// TIA Portal V20 export
// export: Created 2025-12-01T14:56:30.7058292Z, ExportSetting None, DisplayName Totally Integrated Automation Portal, DisplayVersion V20 Update 3, DisplayName TIA Portal Openness, DisplayVersion V20 Update 3, DisplayName TIA Portal Version Control Interface, DisplayVersion V20 Update 3, DisplayName STEP 7 Professional, DisplayVersion V20 Update 3, DisplayName STEP 7 Safety, DisplayVersion V20 Update 2, DisplayName WinCC Basic/Comfort/Advanced, DisplayVersion V20 Update 3, DisplayName WinCC Professional, DisplayVersion V20 Update 3, DisplayName WinCC Unified, DisplayVersion V20 Update 3
FUNCTION_BLOCK "FB435_CRTL_V_E1_S23_BLOQ_OrdJDT"   // FB435, LAD
TITLE = Control del Ramal de Salidas
{ S7_Optimized_Access := 'FALSE' }
AUTHOR : TLigero
NAME : 20190213
VERSION : 3.3
// stored: AutoNumber false, SetENOAutomatically false
   VAR_INPUT
      Mesa : UInt;   // Número de mesa
      En_Tension : Bool;
      pHsMx_E1 : Bool;   // pHs DE PRESENCIA de la Mesa en E1
      pHsMx_S3 : Bool;   // pHs DE AUSENCIA de la Mesa en S3
      pHsMx_S2 : Bool;   // pHs DE AUSENCIA de la Mesa en S2
      En_Pos_WS_0 : Bool;   // Desviador en posicion 0 grados
      En_Pos_WS_45 : Bool;   // Desviador en posicion de desvio
      Termico_E1S3 : Bool;   // Proteccion del Tx en E1E3
      Avance_Tx_Ent : Bool;   // Avance del Tx de entrada. Primer tramo
      Avance_Tx_Sal : Bool;   // Avance del Tx de Salida por S3 o S2
      PTF_Sal_M3 : Bool;   // S3 >> Mesa Siguiente PTF
      NXT_Avance_S3 : Bool;   // S3 >> Mesa Siguiente avanzando
      PTF_Sal_M2 : Bool;   // S2 >> Mesa Siguiente PTF
      NXT_Avance_S2 : Bool;   // S2 >> Mesa Siguiente avanzando
      F_EnvMens_Mx : Bool;   // Fin de Envio de Mensaje
      Mx_Bloq_Activo : Bool;   // Bloqueo Activo de la Mesa
      MX_FlujoPrin_S2 : Bool;   // El flujo principal es Saliendo por S2
      AVTF_MAnt_Mx : Bool;   // E1 >> Mesa Anterior AVTF
      Habilitar_orden_JDT : Bool := false;   // El JDT tendrá el control del cruce con orden
      Num_Cruce : UInt;   // Número de cruce.
      DB_FIFO_Cruce : UInt := 213;   // DB de la FIFO de ordenes del cruce
      Lng_FIFO_Cruce : UInt := 1;   // Longitut de la FIFO de ordenes del cruce
      Valor_Orden_S2 : Word := 16#81;   // Con que orden entra por S2
      MesaS2 : UInt;   // Número de mesa por S2
      MesaS3 : UInt;   // Número de mesa por S3
      V_CNT_pHsMx : UDInt := 500;   // Valor de Presencia en ms
      V_CNT_ApHsMx : UDInt := 500;   // Valor de Ausencia en ms
      V_Vaciado : UDInt := 5000;   // Valor de vaciado en ms
      V_TOut_Desviador : UDInt := 2000;   // TimeOut de los cilindros del desviador en ms
      V_TOut_Tx_Mx : UDInt := 3000;   // TimeOut de Atasco en ms
      V_CNT_ApHsMx_S3 : UDInt := 500;   // Valor de Ausencia por S3 en ms
      V_CNT_ApHsMx_S2 : UDInt := 500;   // Valor de Ausencia por S2 en ms
      V_Orden_Bloqueo : UDInt := 3000;   // en ms
   END_VAR
   VAR_OUTPUT
      P_EnvMens_PMx : Bool;   // Permiso de Enviar Mensaje de Presencia
      Etiqueta_Jdt : UDInt;   // Etiqueta que ha sido leida
      Orden_Ejecutada_Jdt : UInt;   // Orden que se ha ejecutado
      PTF_MAnt_Mx : Bool;   // E1 >> Mesa Anterior PTF
      AVTF_Sal_M2 : Bool;   // S3 >> Mesa Siguiente AVTF
      NXT_Descarga_Act_S2 : Bool;   // S3 >> Mesa Siguiente descarga activa
      AVTF_Sal_M3 : Bool;   // S3 >> Mesa Siguiente AVTF
      NXT_Descarga_Act_S3 : Bool;   // S3 >> Mesa Siguiente descarga activa
   END_VAR
   VAR
      T1_ET00 : Bool;   // Reset
      T1_ET08 : Bool;
      T1_ET01 : Bool;   // Entrada Vacia
      T1_ET10 : Bool;   // Carga Entrada
      T1_ET02 : Bool;   // Entrada Cargada
      T1_ET03 : Bool;   // Vaciando Entrada
      T1_ET20 : Bool;   // Carga Salida
      T1_ET21 : Bool;   // Salida Vacia
      T1_ET50 : Bool;   // Continuar
      T1_ET60 : Bool;   // Entrar
      T1_ET110 : Bool;   // Extraer orden
      T1_ET111 : Bool;
      T1_ET112 : Bool;
      T1_ET02_JDT : Bool;
      FP_ET2_JDT : Bool;
      FIFO_OK : Bool;
      TRANS_OK : Bool;
      O_Bloqueo : Bool;
      Vaciado_1 : Bool;
      Vaciado_2 : Bool;
      FN_ET20 : Bool;
      MemoPresenciaJdt : Bool;
      Maux_FN_Phs_S2 : Bool;
      mem_fn_phs_s2 : Bool;
      Maux_FN_Phs_S3 : Bool;
      mem_fn_phs_s3 : Bool;
      maux_fp_disparo : Bool;
      maux_fn_phs_e1 : Bool;
      ok_vaciado : Bool;
      CNT_ERR_PHS : Int;
      CNT_pHs_WS : UDInt;
      CNT_Aus_WS : UDInt;
      CNT_aus_ent : UDInt;
      CNT_aus_cont : UDInt;
      CNT_bloqueo : UDInt;
      TIMV_WS : UDInt;
      TMP_Err_Pist_pos_0 : UDInt;
      TMP_Paro : UDInt;
      TMP_Err_Pist_pos_45 : UDInt;
      TMP_Err_Tout_avance_E : UDInt;
      TMP_Err_Tout_avance_S : UDInt;
      TMP_En_Tension : UDInt;
      Datos_Scanner { S7_SetPoint := 'True'} : "ROUT_Orden_Fifo_Scanner";
   END_VAR
   VAR_TEMP
      EstadoZona : "EstadoZona";   // Estado de Zona de la Mesa
      EstadoVI : "EstadosMesa";   // Estado del Vehiculo Inteliguente de la Mesa
      ConfigFB : "UDT_ConfigFB";   // Configuracion de la FB de la Mesa
      TEMP_ET00 : Bool;
      O_Continuar : Bool;
      O_Entrar : Bool;
      O_Vaciar : Bool;
      cnt_phs_ok : Bool;
      cnt_aus_ok : Bool;
      OK_Aus_Entrar : Bool;
      OK_Aus_Cont : Bool;
      timeout_piston : Bool;
      ok_tension : Bool;
      Aux_W_Moti : Word;
      Moti_INIC : Bool;
      Moti_ERRO : Bool;
      Moti_NENC : Bool;
      Moti_NORM : Bool;
      ok_bloqueo : Bool;
      O_Continuar_JDT : Bool;
      O_Entrar_JDT : Bool;
      atasco : Bool;
      t_paro : Bool;
      I_V_Ord_Entrar : UInt;
      I_Ord_Filtrada : UInt;
      INT_ORDEN : UInt;
      Aux_W_Orden : Word;
   END_VAR
   VAR_TEMP   // added for the SCL form of the ladder/FBD networks
      _w1 : Bool;
      _w2 : Bool;
      _w3 : Bool;
      _w4 : Bool;
      _w5 : Bool;
      _w6 : Bool;
      _w7 : Bool;
   END_VAR
BEGIN

REGION Network 1: INICIALIZAR - Recoger las Variables de Estado de la Mesa
   // Se recoge - Estado_CBx
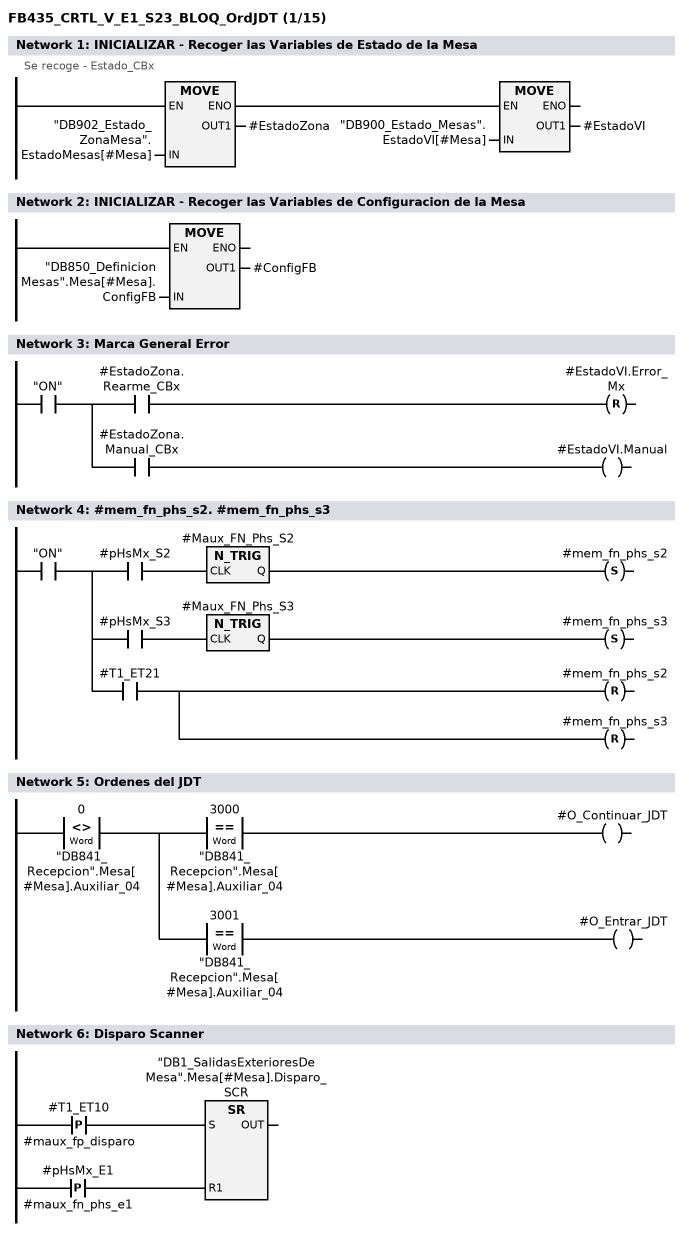
   RUNG wire#powerrail
      Move(in := "DB902_Estado_ZonaMesa".EstadoMesas[#Mesa], out1 => #EstadoZona)
      Move(in := "DB900_Estado_Mesas".EstadoVI[#Mesa], out1 => #EstadoVI)
   END_RUNG
   // the same network as SCL:
   #EstadoZona := "DB902_Estado_ZonaMesa".EstadoMesas[#Mesa];
   #EstadoVI := "DB900_Estado_Mesas".EstadoVI[#Mesa];
END_REGION

REGION Network 2: INICIALIZAR - Recoger las Variables de Configuracion de la Mesa
   RUNG wire#powerrail
      Move(in := "DB850_DefinicionMesas".Mesa[#Mesa].ConfigFB, out1 => #ConfigFB)
   END_RUNG
   // the same network as SCL:
   #ConfigFB := "DB850_DefinicionMesas".Mesa[#Mesa].ConfigFB;
END_REGION

REGION Network 3: Marca General Error
   RUNG wire#powerrail
      Contact( "ON" )
      wire#w1
      Contact( #EstadoZona.Rearme_CBx )
      R_Coil( #EstadoVI.Error_Mx )
   END_RUNG
   RUNG wire#w1
      Contact( #EstadoZona.Manual_CBx )
      Coil( #EstadoVI.Manual )
   END_RUNG
   // the same network as SCL:
   IF "ON" AND #EstadoZona.Rearme_CBx THEN #EstadoVI.Error_Mx := FALSE; END_IF;
   #EstadoVI.Manual := "ON" AND #EstadoZona.Manual_CBx;
END_REGION

REGION Network 4: #mem_fn_phs_s2. #mem_fn_phs_s3
   RUNG wire#powerrail
      Contact( "ON" )
      wire#w1
      Contact( #pHsMx_S2 )
      N_Trig( #Maux_FN_Phs_S2 )
      S_Coil( #mem_fn_phs_s2 )
   END_RUNG
   RUNG wire#w1
      Contact( #pHsMx_S3 )
      N_Trig( #Maux_FN_Phs_S3 )
      S_Coil( #mem_fn_phs_s3 )
   END_RUNG
   RUNG wire#w1
      Contact( #T1_ET21 )
      wire#w2
      R_Coil( #mem_fn_phs_s2 )
   END_RUNG
   RUNG wire#w2
      R_Coil( #mem_fn_phs_s3 )
   END_RUNG
   // the same network as SCL:
   #_w1 := "ON" AND #pHsMx_S2;
   #_w2 := NOT #_w1 AND #Maux_FN_Phs_S2;   // falling edge
   #Maux_FN_Phs_S2 := #_w1;
   IF #_w2 THEN #mem_fn_phs_s2 := TRUE; END_IF;
   #_w3 := "ON" AND #pHsMx_S3;
   #_w4 := NOT #_w3 AND #Maux_FN_Phs_S3;   // falling edge
   #Maux_FN_Phs_S3 := #_w3;
   IF #_w4 THEN #mem_fn_phs_s3 := TRUE; END_IF;
   IF "ON" AND #T1_ET21 THEN
       #mem_fn_phs_s2 := FALSE;
       #mem_fn_phs_s3 := FALSE;
   END_IF;
END_REGION

REGION Network 5: Ordenes del JDT
   RUNG wire#powerrail
      { S7_Templates := "SrcType := Word" } NE_Contact(in1 := 0, in2 := "DB841_Recepcion".Mesa[#Mesa].Auxiliar_04)
      wire#w1
      { S7_Templates := "SrcType := Word" } EQ_Contact(in1 := 3000, in2 := "DB841_Recepcion".Mesa[#Mesa].Auxiliar_04)
      Coil( #O_Continuar_JDT )
   END_RUNG
   RUNG wire#w1
      { S7_Templates := "SrcType := Word" } EQ_Contact(in1 := 3001, in2 := "DB841_Recepcion".Mesa[#Mesa].Auxiliar_04)
      Coil( #O_Entrar_JDT )
   END_RUNG
   // the same network as SCL:
   #_w1 := 0 <> "DB841_Recepcion".Mesa[#Mesa].Auxiliar_04;
   #O_Continuar_JDT := #_w1 AND (3000 = "DB841_Recepcion".Mesa[#Mesa].Auxiliar_04);
   #O_Entrar_JDT := #_w1 AND (3001 = "DB841_Recepcion".Mesa[#Mesa].Auxiliar_04);
END_REGION

REGION Network 6: Disparo Scanner
   RUNG wire#powerrail
      P_Contact(operand := #T1_ET10, bit := #maux_fp_disparo)
      S_SR(operand := "DB1_SalidasExterioresDeMesa".Mesa[#Mesa].Disparo_SCR, r1 := wire#w1)
   END_RUNG
   RUNG wire#powerrail
      P_Contact(operand := #pHsMx_E1, bit := #maux_fn_phs_e1)
   END_RUNG wire#w1
   // the same network as SCL:
   #_w1 := #T1_ET10 AND NOT #maux_fp_disparo;   // rising edge of #T1_ET10
   #maux_fp_disparo := #T1_ET10;
   #_w2 := #pHsMx_E1 AND NOT #maux_fn_phs_e1;   // rising edge of #pHsMx_E1
   #maux_fn_phs_e1 := #pHsMx_E1;
   IF #_w1 THEN
       "DB1_SalidasExterioresDeMesa".Mesa[#Mesa].Disparo_SCR := TRUE;   // SR flip-flop
   END_IF;
   IF #_w2 THEN "DB1_SalidasExterioresDeMesa".Mesa[#Mesa].Disparo_SCR := FALSE; END_IF;
END_REGION

REGION Network 7: GESTION FORZAR ORDENES VACIADO ZONA
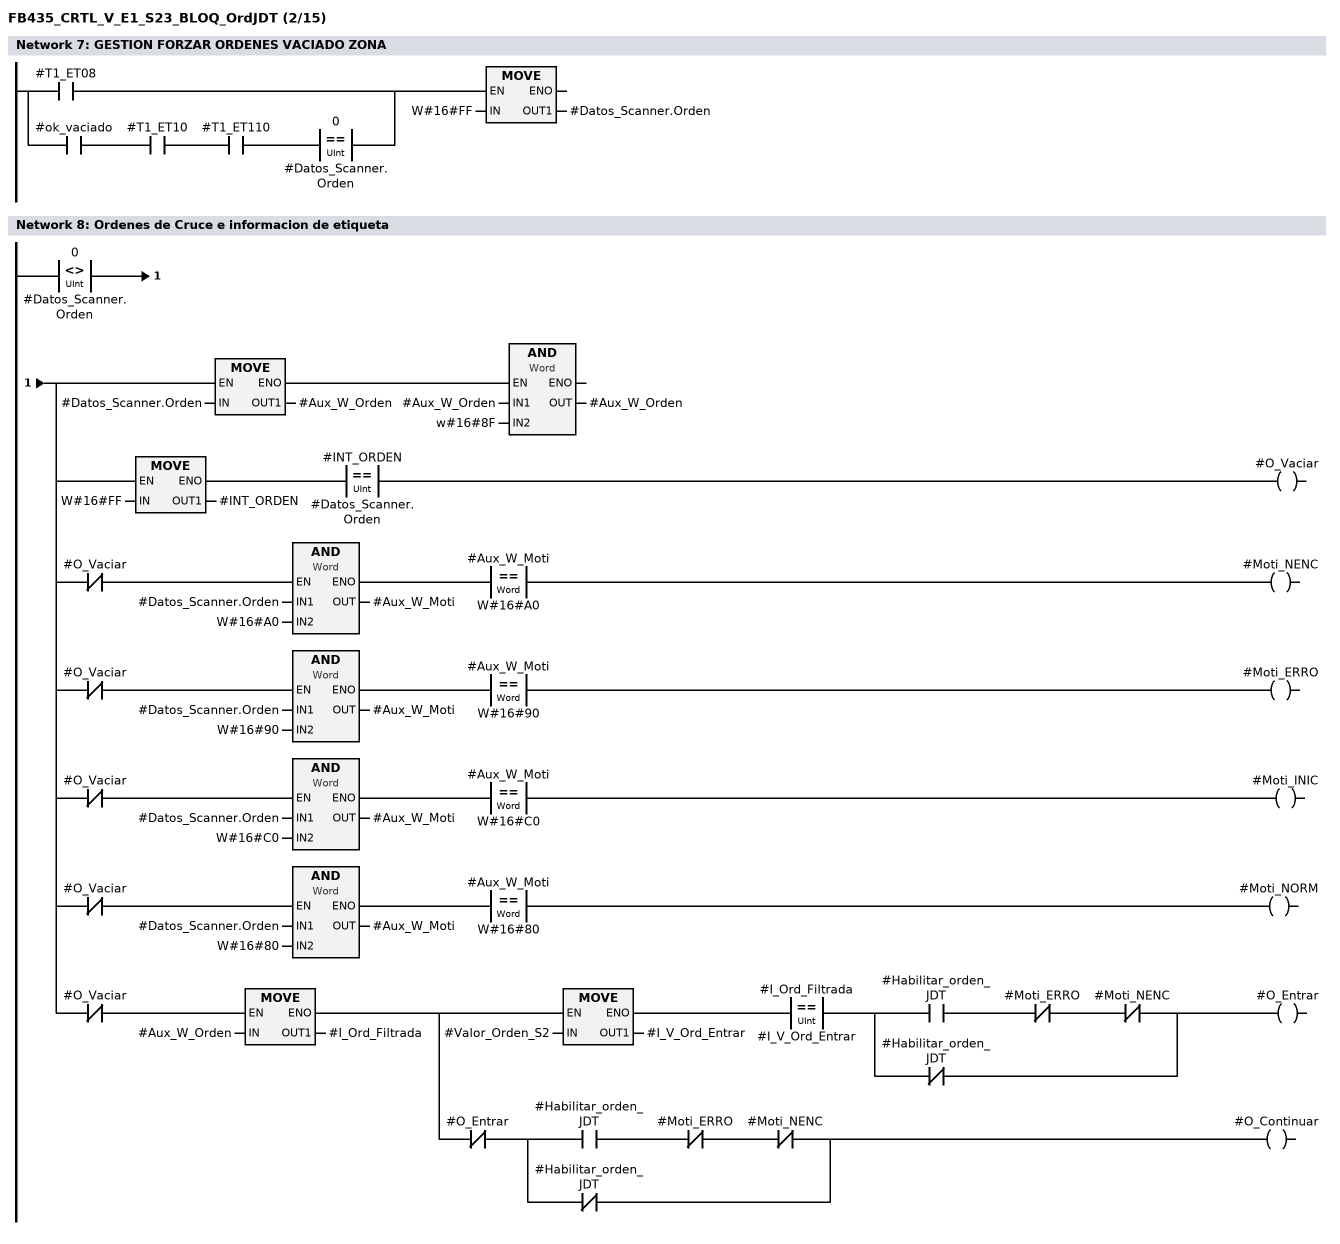
   RUNG wire#powerrail
      Contact( #T1_ET08 )
      wire#w1
      { S7_GenerateENO := "TRUE" } Move(in := W#16#FF, out1 => #Datos_Scanner.Orden)
   END_RUNG
   RUNG wire#powerrail
      Contact( #ok_vaciado )
      Contact( #T1_ET10 )
      Contact( #T1_ET110 )
      { S7_Templates := "SrcType := UInt" } EQ_Contact(in1 := 0, in2 := #Datos_Scanner.Orden)
   END_RUNG wire#w1
   // the same network as SCL:
   IF #T1_ET08 OR (#ok_vaciado AND #T1_ET10 AND #T1_ET110 AND (0 = #Datos_Scanner.Orden)) THEN
       #Datos_Scanner.Orden := W#16#FF;
   END_IF;
END_REGION

REGION Network 8: Ordenes de Cruce e informacion de etiqueta
   RUNG wire#powerrail
      { S7_Templates := "SrcType := UInt" } NE_Contact(in1 := 0, in2 := #Datos_Scanner.Orden)
      wire#w1
      { S7_GenerateENO := "TRUE" } Move(in := #Datos_Scanner.Orden, out1 => #Aux_W_Orden)
      { S7_Templates := "SrcType := Word"; S7_GenerateENO := "TRUE" } And(in1 := #Aux_W_Orden, in2 := w#16#8F, out => #Aux_W_Orden)
   END_RUNG
   RUNG wire#w1
      { S7_GenerateENO := "TRUE" } Move(in := W#16#FF, out1 => #INT_ORDEN)
      { S7_Templates := "SrcType := UInt" } EQ_Contact(in1 := #INT_ORDEN, in2 := #Datos_Scanner.Orden)
      Coil( #O_Vaciar )
   END_RUNG
   RUNG wire#w1
      I_Contact( #O_Vaciar )
      { S7_Templates := "SrcType := Word"; S7_GenerateENO := "TRUE" } And(in1 := #Datos_Scanner.Orden, in2 := W#16#A0, out => #Aux_W_Moti)
      { S7_Templates := "SrcType := Word" } EQ_Contact(in1 := #Aux_W_Moti, in2 := W#16#A0)
      Coil( #Moti_NENC )
   END_RUNG
   RUNG wire#w1
      I_Contact( #O_Vaciar )
      { S7_Templates := "SrcType := Word"; S7_GenerateENO := "TRUE" } And(in1 := #Datos_Scanner.Orden, in2 := W#16#90, out => #Aux_W_Moti)
      { S7_Templates := "SrcType := Word" } EQ_Contact(in1 := #Aux_W_Moti, in2 := W#16#90)
      Coil( #Moti_ERRO )
   END_RUNG
   RUNG wire#w1
      I_Contact( #O_Vaciar )
      { S7_Templates := "SrcType := Word"; S7_GenerateENO := "TRUE" } And(in1 := #Datos_Scanner.Orden, in2 := W#16#C0, out => #Aux_W_Moti)
      { S7_Templates := "SrcType := Word" } EQ_Contact(in1 := #Aux_W_Moti, in2 := W#16#C0)
      Coil( #Moti_INIC )
   END_RUNG
   RUNG wire#w1
      I_Contact( #O_Vaciar )
      { S7_Templates := "SrcType := Word"; S7_GenerateENO := "TRUE" } And(in1 := #Datos_Scanner.Orden, in2 := W#16#80, out => #Aux_W_Moti)
      { S7_Templates := "SrcType := Word" } EQ_Contact(in1 := #Aux_W_Moti, in2 := W#16#80)
      Coil( #Moti_NORM )
   END_RUNG
   RUNG wire#w1
      I_Contact( #O_Vaciar )
      { S7_GenerateENO := "TRUE" } Move(in := #Aux_W_Orden, out1 => #I_Ord_Filtrada)
      wire#w2
      { S7_GenerateENO := "TRUE" } Move(in := #Valor_Orden_S2, out1 => #I_V_Ord_Entrar)
      { S7_Templates := "SrcType := UInt" } EQ_Contact(in1 := #I_Ord_Filtrada, in2 := #I_V_Ord_Entrar)
      wire#w3
      Contact( #Habilitar_orden_JDT )
      I_Contact( #Moti_ERRO )
      I_Contact( #Moti_NENC )
      wire#w4
      Coil( #O_Entrar )
   END_RUNG
   RUNG wire#w3
      I_Contact( #Habilitar_orden_JDT )
   END_RUNG wire#w4
   RUNG wire#w2
      I_Contact( #O_Entrar )
      wire#w5
      Contact( #Habilitar_orden_JDT )
      I_Contact( #Moti_ERRO )
      I_Contact( #Moti_NENC )
      wire#w6
      Coil( #O_Continuar )
   END_RUNG
   RUNG wire#w5
      I_Contact( #Habilitar_orden_JDT )
   END_RUNG wire#w6
   // the same network as SCL:
   // ENO of a box is taken as its EN; it also drops when the box reports an error
   #_w1 := 0 <> #Datos_Scanner.Orden;
   IF #_w1 THEN
       #Aux_W_Orden := #Datos_Scanner.Orden;
       #Aux_W_Orden := #Aux_W_Orden AND w#16#8F;
       #INT_ORDEN := W#16#FF;
   END_IF;
   #O_Vaciar := #_w1 AND (#INT_ORDEN = #Datos_Scanner.Orden);
   #_w2 := #_w1 AND NOT #O_Vaciar;
   IF #_w2 THEN #Aux_W_Moti := #Datos_Scanner.Orden AND W#16#A0; END_IF;
   #Moti_NENC := #_w2 AND (#Aux_W_Moti = W#16#A0);
   #_w3 := #_w1 AND NOT #O_Vaciar;
   IF #_w3 THEN #Aux_W_Moti := #Datos_Scanner.Orden AND W#16#90; END_IF;
   #Moti_ERRO := #_w3 AND (#Aux_W_Moti = W#16#90);
   #_w4 := #_w1 AND NOT #O_Vaciar;
   IF #_w4 THEN #Aux_W_Moti := #Datos_Scanner.Orden AND W#16#C0; END_IF;
   #Moti_INIC := #_w4 AND (#Aux_W_Moti = W#16#C0);
   #_w5 := #_w1 AND NOT #O_Vaciar;
   IF #_w5 THEN #Aux_W_Moti := #Datos_Scanner.Orden AND W#16#80; END_IF;
   #Moti_NORM := #_w5 AND (#Aux_W_Moti = W#16#80);
   #_w6 := #_w1 AND NOT #O_Vaciar;
   IF #_w6 THEN
       #I_Ord_Filtrada := #Aux_W_Orden;
       #I_V_Ord_Entrar := #Valor_Orden_S2;
   END_IF;
   #O_Entrar := #_w6 AND (#I_Ord_Filtrada = #I_V_Ord_Entrar) AND ((#Habilitar_orden_JDT AND NOT #Moti_ERRO AND NOT #Moti_NENC) OR NOT #Habilitar_orden_JDT);
   #O_Continuar := #_w6 AND NOT #O_Entrar AND ((#Habilitar_orden_JDT AND NOT #Moti_ERRO AND NOT #Moti_NENC) OR NOT #Habilitar_orden_JDT);
END_REGION

REGION Network 9: FC912. #V_CNTpHsWS
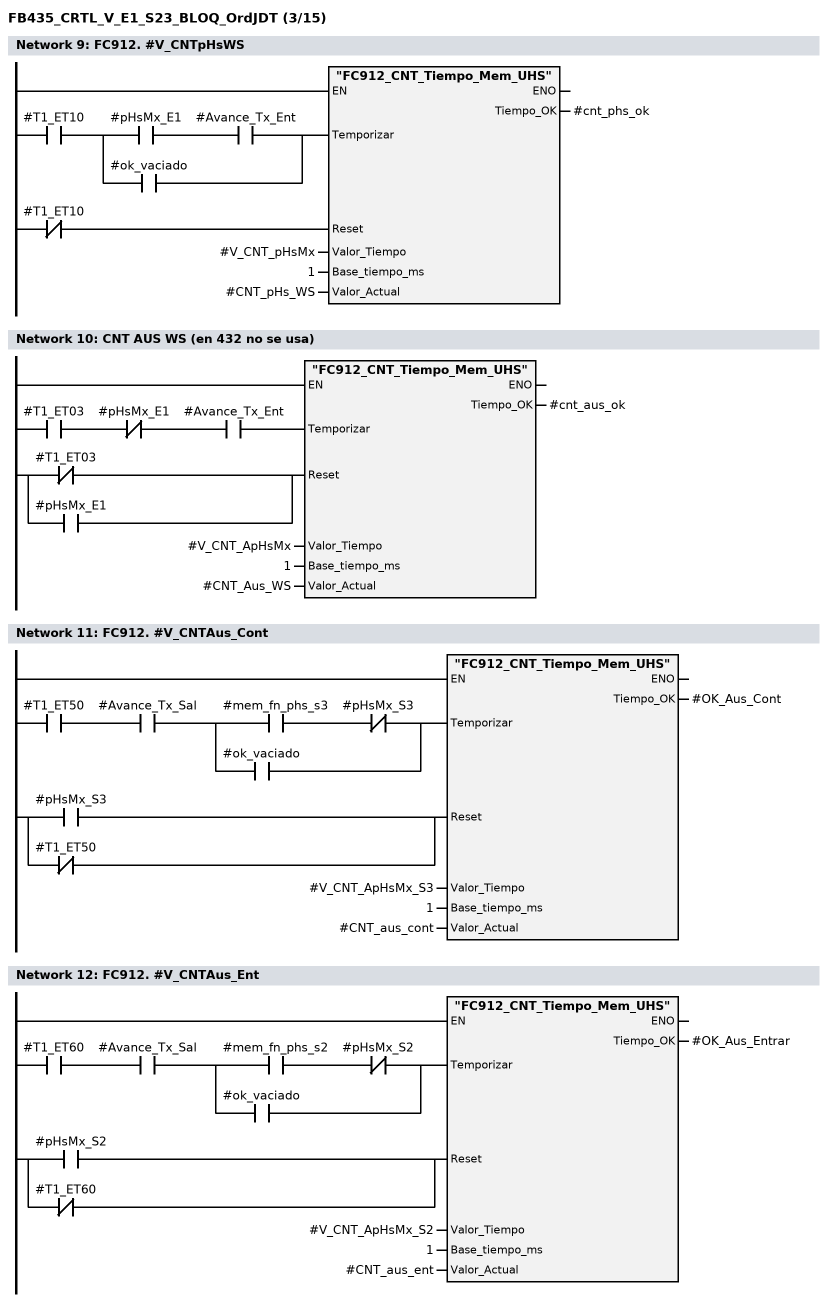
   RUNG wire#powerrail
      "FC912_CNT_Tiempo_Mem_UHS"(Temporizar := wire#w2, Reset := wire#w3, Valor_Tiempo := #V_CNT_pHsMx, Base_tiempo_ms := 1, Valor_Actual := #CNT_pHs_WS, Tiempo_OK => #cnt_phs_ok)
   END_RUNG
   RUNG wire#powerrail
      Contact( #T1_ET10 )
      wire#w1
      Contact( #pHsMx_E1 )
      Contact( #Avance_Tx_Ent )
   END_RUNG wire#w2
   RUNG wire#w1
      Contact( #ok_vaciado )
   END_RUNG wire#w2
   RUNG wire#powerrail
      I_Contact( #T1_ET10 )
   END_RUNG wire#w3
   // the same network as SCL:
   "FC912_CNT_Tiempo_Mem_UHS"(Temporizar := #T1_ET10 AND ((#pHsMx_E1 AND #Avance_Tx_Ent) OR #ok_vaciado),
                           Reset := NOT #T1_ET10,
                           Valor_Tiempo := #V_CNT_pHsMx,
                           Base_tiempo_ms := 1,
                           Valor_Actual := #CNT_pHs_WS,
                           Tiempo_OK => #cnt_phs_ok);
END_REGION

REGION Network 10: CNT AUS WS (en 432 no se usa)
   RUNG wire#powerrail
      "FC912_CNT_Tiempo_Mem_UHS"(Temporizar := wire#w1, Reset := wire#w2, Valor_Tiempo := #V_CNT_ApHsMx, Base_tiempo_ms := 1, Valor_Actual := #CNT_Aus_WS, Tiempo_OK => #cnt_aus_ok)
   END_RUNG
   RUNG wire#powerrail
      Contact( #T1_ET03 )
      I_Contact( #pHsMx_E1 )
      Contact( #Avance_Tx_Ent )
   END_RUNG wire#w1
   RUNG wire#powerrail
      I_Contact( #T1_ET03 )
   END_RUNG wire#w2
   RUNG wire#powerrail
      Contact( #pHsMx_E1 )
   END_RUNG wire#w2
   // the same network as SCL:
   "FC912_CNT_Tiempo_Mem_UHS"(Temporizar := #T1_ET03 AND NOT #pHsMx_E1 AND #Avance_Tx_Ent,
                           Reset := NOT #T1_ET03 OR #pHsMx_E1,
                           Valor_Tiempo := #V_CNT_ApHsMx,
                           Base_tiempo_ms := 1,
                           Valor_Actual := #CNT_Aus_WS,
                           Tiempo_OK => #cnt_aus_ok);
END_REGION

REGION Network 11: FC912. #V_CNTAus_Cont
   RUNG wire#powerrail
      "FC912_CNT_Tiempo_Mem_UHS"(Temporizar := wire#w2, Reset := wire#w3, Valor_Tiempo := #V_CNT_ApHsMx_S3, Base_tiempo_ms := 1, Valor_Actual := #CNT_aus_cont, Tiempo_OK => #OK_Aus_Cont)
   END_RUNG
   RUNG wire#powerrail
      Contact( #T1_ET50 )
      Contact( #Avance_Tx_Sal )
      wire#w1
      Contact( #mem_fn_phs_s3 )
      I_Contact( #pHsMx_S3 )
   END_RUNG wire#w2
   RUNG wire#w1
      Contact( #ok_vaciado )
   END_RUNG wire#w2
   RUNG wire#powerrail
      Contact( #pHsMx_S3 )
   END_RUNG wire#w3
   RUNG wire#powerrail
      I_Contact( #T1_ET50 )
   END_RUNG wire#w3
   // the same network as SCL:
   "FC912_CNT_Tiempo_Mem_UHS"(Temporizar := #T1_ET50 AND #Avance_Tx_Sal AND ((#mem_fn_phs_s3 AND NOT #pHsMx_S3) OR #ok_vaciado),
                           Reset := #pHsMx_S3 OR NOT #T1_ET50,
                           Valor_Tiempo := #V_CNT_ApHsMx_S3,
                           Base_tiempo_ms := 1,
                           Valor_Actual := #CNT_aus_cont,
                           Tiempo_OK => #OK_Aus_Cont);
END_REGION

REGION Network 12: FC912. #V_CNTAus_Ent
   RUNG wire#powerrail
      "FC912_CNT_Tiempo_Mem_UHS"(Temporizar := wire#w2, Reset := wire#w3, Valor_Tiempo := #V_CNT_ApHsMx_S2, Base_tiempo_ms := 1, Valor_Actual := #CNT_aus_ent, Tiempo_OK => #OK_Aus_Entrar)
   END_RUNG
   RUNG wire#powerrail
      Contact( #T1_ET60 )
      Contact( #Avance_Tx_Sal )
      wire#w1
      Contact( #mem_fn_phs_s2 )
      I_Contact( #pHsMx_S2 )
   END_RUNG wire#w2
   RUNG wire#w1
      Contact( #ok_vaciado )
   END_RUNG wire#w2
   RUNG wire#powerrail
      Contact( #pHsMx_S2 )
   END_RUNG wire#w3
   RUNG wire#powerrail
      I_Contact( #T1_ET60 )
   END_RUNG wire#w3
   // the same network as SCL:
   "FC912_CNT_Tiempo_Mem_UHS"(Temporizar := #T1_ET60 AND #Avance_Tx_Sal AND ((#mem_fn_phs_s2 AND NOT #pHsMx_S2) OR #ok_vaciado),
                           Reset := #pHsMx_S2 OR NOT #T1_ET60,
                           Valor_Tiempo := #V_CNT_ApHsMx_S2,
                           Base_tiempo_ms := 1,
                           Valor_Actual := #CNT_aus_ent,
                           Tiempo_OK => #OK_Aus_Entrar);
END_REGION

REGION Network 13: FC912. #V_TmpBloqueo
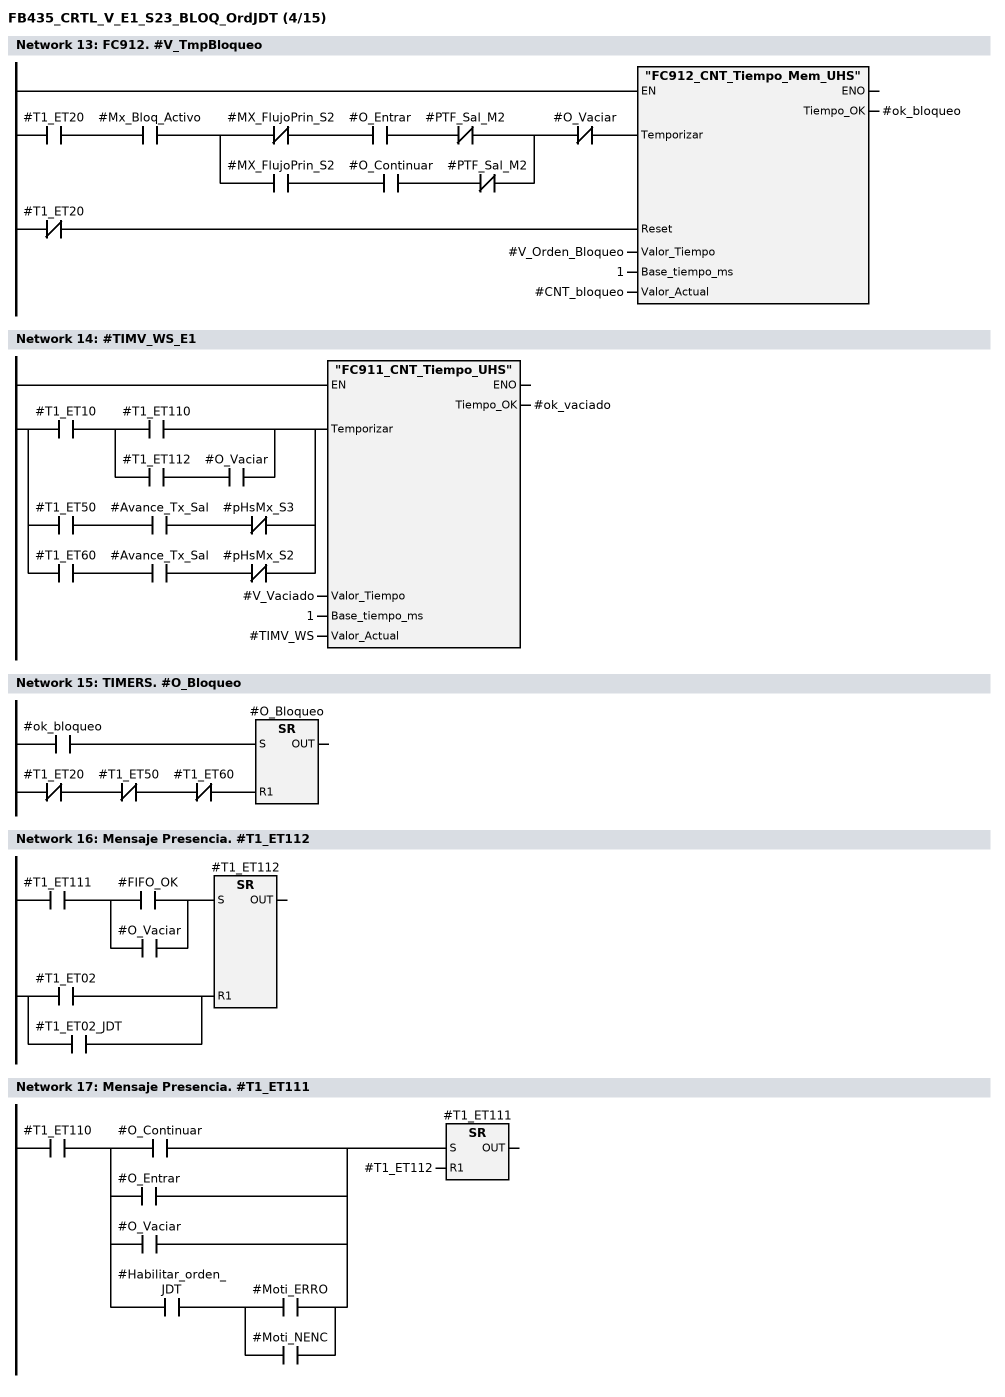
   RUNG wire#powerrail
      "FC912_CNT_Tiempo_Mem_UHS"(Temporizar := wire#w3, Reset := wire#w4, Valor_Tiempo := #V_Orden_Bloqueo, Base_tiempo_ms := 1, Valor_Actual := #CNT_bloqueo, Tiempo_OK => #ok_bloqueo)
   END_RUNG
   RUNG wire#powerrail
      Contact( #T1_ET20 )
      Contact( #Mx_Bloq_Activo )
      wire#w1
      I_Contact( #MX_FlujoPrin_S2 )
      Contact( #O_Entrar )
      I_Contact( #PTF_Sal_M2 )
      wire#w2
      I_Contact( #O_Vaciar )
   END_RUNG wire#w3
   RUNG wire#w1
      Contact( #MX_FlujoPrin_S2 )
      Contact( #O_Continuar )
      I_Contact( #PTF_Sal_M2 )
   END_RUNG wire#w2
   RUNG wire#powerrail
      I_Contact( #T1_ET20 )
   END_RUNG wire#w4
   // the same network as SCL:
   "FC912_CNT_Tiempo_Mem_UHS"(Temporizar := #T1_ET20 AND #Mx_Bloq_Activo AND ((NOT #MX_FlujoPrin_S2 AND #O_Entrar AND NOT #PTF_Sal_M2) OR (#MX_FlujoPrin_S2 AND #O_Continuar AND NOT #PTF_Sal_M2)) AND NOT #O_Vaciar,
                           Reset := NOT #T1_ET20,
                           Valor_Tiempo := #V_Orden_Bloqueo,
                           Base_tiempo_ms := 1,
                           Valor_Actual := #CNT_bloqueo,
                           Tiempo_OK => #ok_bloqueo);
END_REGION

REGION Network 14: #TIMV_WS_E1
   RUNG wire#powerrail
      "FC911_CNT_Tiempo_UHS"(Temporizar := wire#w2, Valor_Tiempo := #V_Vaciado, Base_tiempo_ms := 1, Valor_Actual := #TIMV_WS, Tiempo_OK => #ok_vaciado)
   END_RUNG
   RUNG wire#powerrail
      Contact( #T1_ET10 )
      wire#w1
      Contact( #T1_ET110 )
   END_RUNG wire#w2
   RUNG wire#w1
      Contact( #T1_ET112 )
      Contact( #O_Vaciar )
   END_RUNG wire#w2
   RUNG wire#powerrail
      Contact( #T1_ET50 )
      Contact( #Avance_Tx_Sal )
      I_Contact( #pHsMx_S3 )
   END_RUNG wire#w2
   RUNG wire#powerrail
      Contact( #T1_ET60 )
      Contact( #Avance_Tx_Sal )
      I_Contact( #pHsMx_S2 )
   END_RUNG wire#w2
   // the same network as SCL:
   "FC911_CNT_Tiempo_UHS"(Temporizar := (#T1_ET10 AND (#T1_ET110 OR (#T1_ET112 AND #O_Vaciar))) OR (#T1_ET50 AND #Avance_Tx_Sal AND NOT #pHsMx_S3) OR (#T1_ET60 AND #Avance_Tx_Sal AND NOT #pHsMx_S2),
                          Valor_Tiempo := #V_Vaciado,
                          Base_tiempo_ms := 1,
                          Valor_Actual := #TIMV_WS,
                          Tiempo_OK => #ok_vaciado);
END_REGION

REGION Network 15: TIMERS. #O_Bloqueo
   RUNG wire#powerrail
      Contact( #ok_bloqueo )
      S_SR(operand := #O_Bloqueo, r1 := wire#w1)
   END_RUNG
   RUNG wire#powerrail
      I_Contact( #T1_ET20 )
      I_Contact( #T1_ET50 )
      I_Contact( #T1_ET60 )
   END_RUNG wire#w1
   // the same network as SCL:
   IF #ok_bloqueo THEN
       #O_Bloqueo := TRUE;   // SR flip-flop
   END_IF;
   IF NOT #T1_ET20 AND NOT #T1_ET50 AND NOT #T1_ET60 THEN #O_Bloqueo := FALSE; END_IF;
END_REGION

REGION Network 16: Mensaje Presencia. #T1_ET112
   RUNG wire#powerrail
      Contact( #T1_ET111 )
      wire#w1
      Contact( #FIFO_OK )
      wire#w2
      S_SR(operand := #T1_ET112, r1 := wire#w3)
   END_RUNG
   RUNG wire#w1
      Contact( #O_Vaciar )
   END_RUNG wire#w2
   RUNG wire#powerrail
      Contact( #T1_ET02 )
   END_RUNG wire#w3
   RUNG wire#powerrail
      Contact( #T1_ET02_JDT )
   END_RUNG wire#w3
   // the same network as SCL:
   IF #T1_ET111 AND (#FIFO_OK OR #O_Vaciar) THEN
       #T1_ET112 := TRUE;   // SR flip-flop
   END_IF;
   IF #T1_ET02 OR #T1_ET02_JDT THEN #T1_ET112 := FALSE; END_IF;
END_REGION

REGION Network 17: Mensaje Presencia. #T1_ET111
   RUNG wire#powerrail
      Contact( #T1_ET110 )
      wire#w1
      Contact( #O_Continuar )
      wire#w2
      S_SR(operand := #T1_ET111, r1 := #T1_ET112)
   END_RUNG
   RUNG wire#w1
      Contact( #O_Entrar )
   END_RUNG wire#w2
   RUNG wire#w1
      Contact( #O_Vaciar )
   END_RUNG wire#w2
   RUNG wire#w1
      Contact( #Habilitar_orden_JDT )
      wire#w3
      Contact( #Moti_ERRO )
   END_RUNG wire#w2
   RUNG wire#w3
      Contact( #Moti_NENC )
   END_RUNG wire#w2
   // the same network as SCL:
   IF #T1_ET110 AND (#O_Continuar OR #O_Entrar OR #O_Vaciar OR (#Habilitar_orden_JDT AND (#Moti_ERRO OR #Moti_NENC))) THEN
       #T1_ET111 := TRUE;   // SR flip-flop
   END_IF;
   IF #T1_ET112 THEN #T1_ET111 := FALSE; END_IF;
END_REGION

REGION Network 18: #T1_ET110
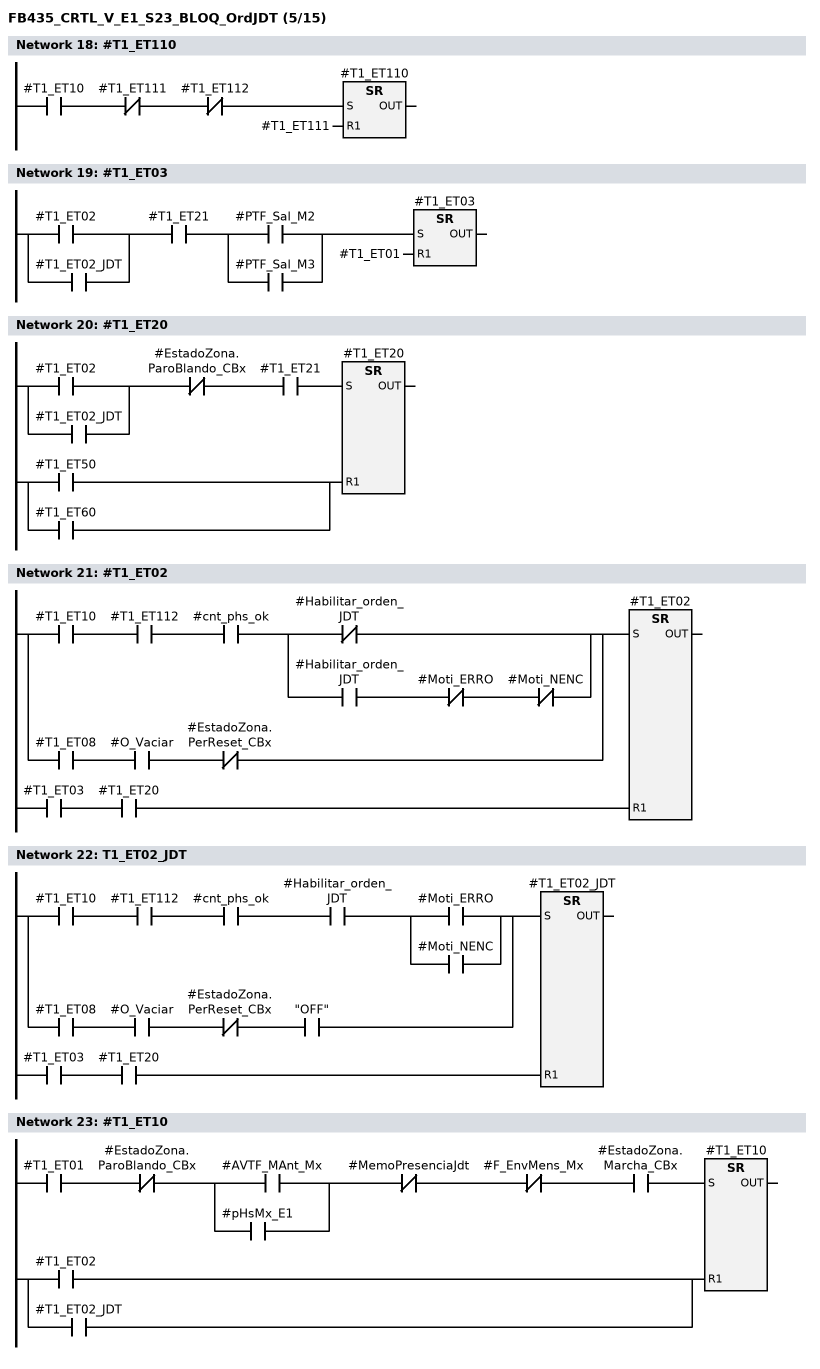
   RUNG wire#powerrail
      Contact( #T1_ET10 )
      I_Contact( #T1_ET111 )
      I_Contact( #T1_ET112 )
      S_SR(operand := #T1_ET110, r1 := #T1_ET111)
   END_RUNG
   // the same network as SCL:
   IF #T1_ET10 AND NOT #T1_ET111 AND NOT #T1_ET112 THEN
       #T1_ET110 := TRUE;   // SR flip-flop
   END_IF;
   IF #T1_ET111 THEN #T1_ET110 := FALSE; END_IF;
END_REGION

REGION Network 19: #T1_ET03
   RUNG wire#powerrail
      Contact( #T1_ET02 )
      wire#w1
      Contact( #T1_ET21 )
      wire#w2
      Contact( #PTF_Sal_M2 )
      wire#w3
      S_SR(operand := #T1_ET03, r1 := #T1_ET01)
   END_RUNG
   RUNG wire#powerrail
      Contact( #T1_ET02_JDT )
   END_RUNG wire#w1
   RUNG wire#w2
      Contact( #PTF_Sal_M3 )
   END_RUNG wire#w3
   // the same network as SCL:
   IF (#T1_ET02 OR #T1_ET02_JDT) AND #T1_ET21 AND (#PTF_Sal_M2 OR #PTF_Sal_M3) THEN
       #T1_ET03 := TRUE;   // SR flip-flop
   END_IF;
   IF #T1_ET01 THEN #T1_ET03 := FALSE; END_IF;
END_REGION

REGION Network 20: #T1_ET20
   RUNG wire#powerrail
      Contact( #T1_ET02 )
      wire#w1
      I_Contact( #EstadoZona.ParoBlando_CBx )
      Contact( #T1_ET21 )
      S_SR(operand := #T1_ET20, r1 := wire#w2)
   END_RUNG
   RUNG wire#powerrail
      Contact( #T1_ET02_JDT )
   END_RUNG wire#w1
   RUNG wire#powerrail
      Contact( #T1_ET50 )
   END_RUNG wire#w2
   RUNG wire#powerrail
      Contact( #T1_ET60 )
   END_RUNG wire#w2
   // the same network as SCL:
   IF (#T1_ET02 OR #T1_ET02_JDT) AND NOT #EstadoZona.ParoBlando_CBx AND #T1_ET21 THEN
       #T1_ET20 := TRUE;   // SR flip-flop
   END_IF;
   IF #T1_ET50 OR #T1_ET60 THEN #T1_ET20 := FALSE; END_IF;
END_REGION

REGION Network 21: #T1_ET02
   RUNG wire#powerrail
      Contact( #T1_ET10 )
      Contact( #T1_ET112 )
      Contact( #cnt_phs_ok )
      wire#w1
      I_Contact( #Habilitar_orden_JDT )
      wire#w2
      S_SR(operand := #T1_ET02, r1 := wire#w3)
   END_RUNG
   RUNG wire#w1
      Contact( #Habilitar_orden_JDT )
      I_Contact( #Moti_ERRO )
      I_Contact( #Moti_NENC )
   END_RUNG wire#w2
   RUNG wire#powerrail
      Contact( #T1_ET08 )
      Contact( #O_Vaciar )
      I_Contact( #EstadoZona.PerReset_CBx )
   END_RUNG wire#w2
   RUNG wire#powerrail
      Contact( #T1_ET03 )
      Contact( #T1_ET20 )
   END_RUNG wire#w3
   // the same network as SCL:
   IF (#T1_ET10 AND #T1_ET112 AND #cnt_phs_ok AND (NOT #Habilitar_orden_JDT OR (#Habilitar_orden_JDT AND NOT #Moti_ERRO AND NOT #Moti_NENC))) OR (#T1_ET08 AND #O_Vaciar AND NOT #EstadoZona.PerReset_CBx) THEN
       #T1_ET02 := TRUE;   // SR flip-flop
   END_IF;
   IF #T1_ET03 AND #T1_ET20 THEN #T1_ET02 := FALSE; END_IF;
END_REGION

REGION Network 22: T1_ET02_JDT
   RUNG wire#powerrail
      Contact( #T1_ET10 )
      Contact( #T1_ET112 )
      Contact( #cnt_phs_ok )
      Contact( #Habilitar_orden_JDT )
      wire#w1
      Contact( #Moti_ERRO )
      wire#w2
      S_SR(operand := #T1_ET02_JDT, r1 := wire#w3)
   END_RUNG
   RUNG wire#w1
      Contact( #Moti_NENC )
   END_RUNG wire#w2
   RUNG wire#powerrail
      Contact( #T1_ET08 )
      Contact( #O_Vaciar )
      I_Contact( #EstadoZona.PerReset_CBx )
      Contact( "OFF" )
   END_RUNG wire#w2
   RUNG wire#powerrail
      Contact( #T1_ET03 )
      Contact( #T1_ET20 )
   END_RUNG wire#w3
   // the same network as SCL:
   IF (#T1_ET10 AND #T1_ET112 AND #cnt_phs_ok AND #Habilitar_orden_JDT AND (#Moti_ERRO OR #Moti_NENC)) OR (#T1_ET08 AND #O_Vaciar AND NOT #EstadoZona.PerReset_CBx AND "OFF") THEN
       #T1_ET02_JDT := TRUE;   // SR flip-flop
   END_IF;
   IF #T1_ET03 AND #T1_ET20 THEN #T1_ET02_JDT := FALSE; END_IF;
END_REGION

REGION Network 23: #T1_ET10
   RUNG wire#powerrail
      Contact( #T1_ET01 )
      I_Contact( #EstadoZona.ParoBlando_CBx )
      wire#w1
      Contact( #AVTF_MAnt_Mx )
      wire#w2
      I_Contact( #MemoPresenciaJdt )
      I_Contact( #F_EnvMens_Mx )
      Contact( #EstadoZona.Marcha_CBx )
      S_SR(operand := #T1_ET10, r1 := wire#w3)
   END_RUNG
   RUNG wire#w1
      Contact( #pHsMx_E1 )
   END_RUNG wire#w2
   RUNG wire#powerrail
      Contact( #T1_ET02 )
   END_RUNG wire#w3
   RUNG wire#powerrail
      Contact( #T1_ET02_JDT )
   END_RUNG wire#w3
   // the same network as SCL:
   IF #T1_ET01 AND NOT #EstadoZona.ParoBlando_CBx AND (#AVTF_MAnt_Mx OR #pHsMx_E1) AND NOT #MemoPresenciaJdt AND NOT #F_EnvMens_Mx AND #EstadoZona.Marcha_CBx THEN
       #T1_ET10 := TRUE;   // SR flip-flop
   END_IF;
   IF #T1_ET02 OR #T1_ET02_JDT THEN #T1_ET10 := FALSE; END_IF;
END_REGION

REGION Network 24: #T1_ET01
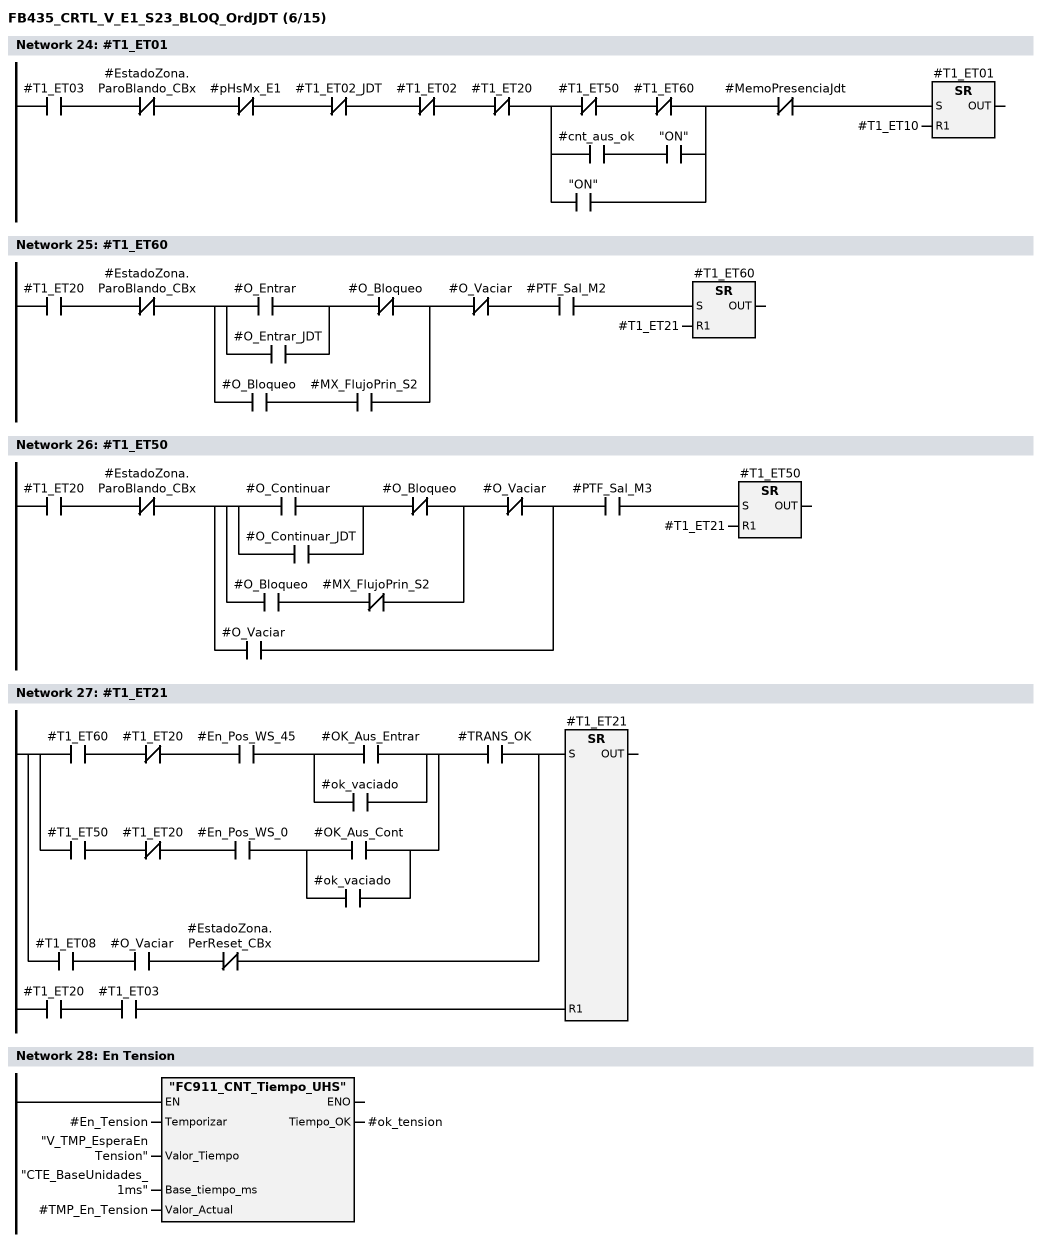
   RUNG wire#powerrail
      Contact( #T1_ET03 )
      I_Contact( #EstadoZona.ParoBlando_CBx )
      I_Contact( #pHsMx_E1 )
      I_Contact( #T1_ET02_JDT )
      I_Contact( #T1_ET02 )
      I_Contact( #T1_ET20 )
      wire#w1
      I_Contact( #T1_ET50 )
      I_Contact( #T1_ET60 )
      wire#w2
      I_Contact( #MemoPresenciaJdt )
      S_SR(operand := #T1_ET01, r1 := #T1_ET10)
   END_RUNG
   RUNG wire#w1
      Contact( #cnt_aus_ok )
      Contact( "ON" )
   END_RUNG wire#w2
   RUNG wire#w1
      Contact( "ON" )
   END_RUNG wire#w2
   // the same network as SCL:
   IF #T1_ET03 AND NOT #EstadoZona.ParoBlando_CBx AND NOT #pHsMx_E1 AND NOT #T1_ET02_JDT AND NOT #T1_ET02 AND NOT #T1_ET20 AND ((NOT #T1_ET50 AND NOT #T1_ET60) OR (#cnt_aus_ok AND "ON") OR "ON") AND NOT #MemoPresenciaJdt THEN
       #T1_ET01 := TRUE;   // SR flip-flop
   END_IF;
   IF #T1_ET10 THEN #T1_ET01 := FALSE; END_IF;
END_REGION

REGION Network 25: #T1_ET60
   RUNG wire#powerrail
      Contact( #T1_ET20 )
      I_Contact( #EstadoZona.ParoBlando_CBx )
      wire#w1
      Contact( #O_Entrar )
      wire#w2
      I_Contact( #O_Bloqueo )
      wire#w3
      I_Contact( #O_Vaciar )
      Contact( #PTF_Sal_M2 )
      S_SR(operand := #T1_ET60, r1 := #T1_ET21)
   END_RUNG
   RUNG wire#w1
      Contact( #O_Entrar_JDT )
   END_RUNG wire#w2
   RUNG wire#w1
      Contact( #O_Bloqueo )
      Contact( #MX_FlujoPrin_S2 )
   END_RUNG wire#w3
   // the same network as SCL:
   IF #T1_ET20 AND NOT #EstadoZona.ParoBlando_CBx AND (((#O_Entrar OR #O_Entrar_JDT) AND NOT #O_Bloqueo) OR (#O_Bloqueo AND #MX_FlujoPrin_S2)) AND NOT #O_Vaciar AND #PTF_Sal_M2 THEN
       #T1_ET60 := TRUE;   // SR flip-flop
   END_IF;
   IF #T1_ET21 THEN #T1_ET60 := FALSE; END_IF;
END_REGION

REGION Network 26: #T1_ET50
   RUNG wire#powerrail
      Contact( #T1_ET20 )
      I_Contact( #EstadoZona.ParoBlando_CBx )
      wire#w1
      Contact( #O_Continuar )
      wire#w2
      I_Contact( #O_Bloqueo )
      wire#w3
      I_Contact( #O_Vaciar )
      wire#w4
      Contact( #PTF_Sal_M3 )
      S_SR(operand := #T1_ET50, r1 := #T1_ET21)
   END_RUNG
   RUNG wire#w1
      Contact( #O_Continuar_JDT )
   END_RUNG wire#w2
   RUNG wire#w1
      Contact( #O_Bloqueo )
      I_Contact( #MX_FlujoPrin_S2 )
   END_RUNG wire#w3
   RUNG wire#w1
      Contact( #O_Vaciar )
   END_RUNG wire#w4
   // the same network as SCL:
   IF #T1_ET20 AND NOT #EstadoZona.ParoBlando_CBx AND (((((#O_Continuar OR #O_Continuar_JDT) AND NOT #O_Bloqueo) OR (#O_Bloqueo AND NOT #MX_FlujoPrin_S2)) AND NOT #O_Vaciar) OR #O_Vaciar) AND #PTF_Sal_M3 THEN
       #T1_ET50 := TRUE;   // SR flip-flop
   END_IF;
   IF #T1_ET21 THEN #T1_ET50 := FALSE; END_IF;
END_REGION

REGION Network 27: #T1_ET21
   RUNG wire#powerrail
      Contact( #T1_ET60 )
      I_Contact( #T1_ET20 )
      Contact( #En_Pos_WS_45 )
      wire#w1
      Contact( #OK_Aus_Entrar )
      wire#w2
      Contact( #TRANS_OK )
      wire#w4
      S_SR(operand := #T1_ET21, r1 := wire#w5)
   END_RUNG
   RUNG wire#w1
      Contact( #ok_vaciado )
   END_RUNG wire#w2
   RUNG wire#powerrail
      Contact( #T1_ET50 )
      I_Contact( #T1_ET20 )
      Contact( #En_Pos_WS_0 )
      wire#w3
      Contact( #OK_Aus_Cont )
   END_RUNG wire#w2
   RUNG wire#w3
      Contact( #ok_vaciado )
   END_RUNG wire#w2
   RUNG wire#powerrail
      Contact( #T1_ET08 )
      Contact( #O_Vaciar )
      I_Contact( #EstadoZona.PerReset_CBx )
   END_RUNG wire#w4
   RUNG wire#powerrail
      Contact( #T1_ET20 )
      Contact( #T1_ET03 )
   END_RUNG wire#w5
   // the same network as SCL:
   IF (((#T1_ET60 AND NOT #T1_ET20 AND #En_Pos_WS_45 AND (#OK_Aus_Entrar OR #ok_vaciado)) OR (#T1_ET50 AND NOT #T1_ET20 AND #En_Pos_WS_0 AND (#OK_Aus_Cont OR #ok_vaciado))) AND #TRANS_OK) OR (#T1_ET08 AND #O_Vaciar AND NOT #EstadoZona.PerReset_CBx) THEN
       #T1_ET21 := TRUE;   // SR flip-flop
   END_IF;
   IF #T1_ET20 AND #T1_ET03 THEN #T1_ET21 := FALSE; END_IF;
END_REGION

REGION Network 28: En Tension
   RUNG wire#powerrail
      "FC911_CNT_Tiempo_UHS"(Temporizar := #En_Tension, Valor_Tiempo := "V_TMP_EsperaEnTension", Base_tiempo_ms := "CTE_BaseUnidades_1ms", Valor_Actual := #TMP_En_Tension, Tiempo_OK => #ok_tension)
   END_RUNG
   // the same network as SCL:
   "FC911_CNT_Tiempo_UHS"(Temporizar := #En_Tension,
                          Valor_Tiempo := "V_TMP_EsperaEnTension",
                          Base_tiempo_ms := "CTE_BaseUnidades_1ms",
                          Valor_Actual := #TMP_En_Tension,
                          Tiempo_OK => #ok_tension);
END_REGION

REGION Network 29: Marca General Error. "DB900_Estado_Mesas".EstadoVI[numeromesa].En_Termico1
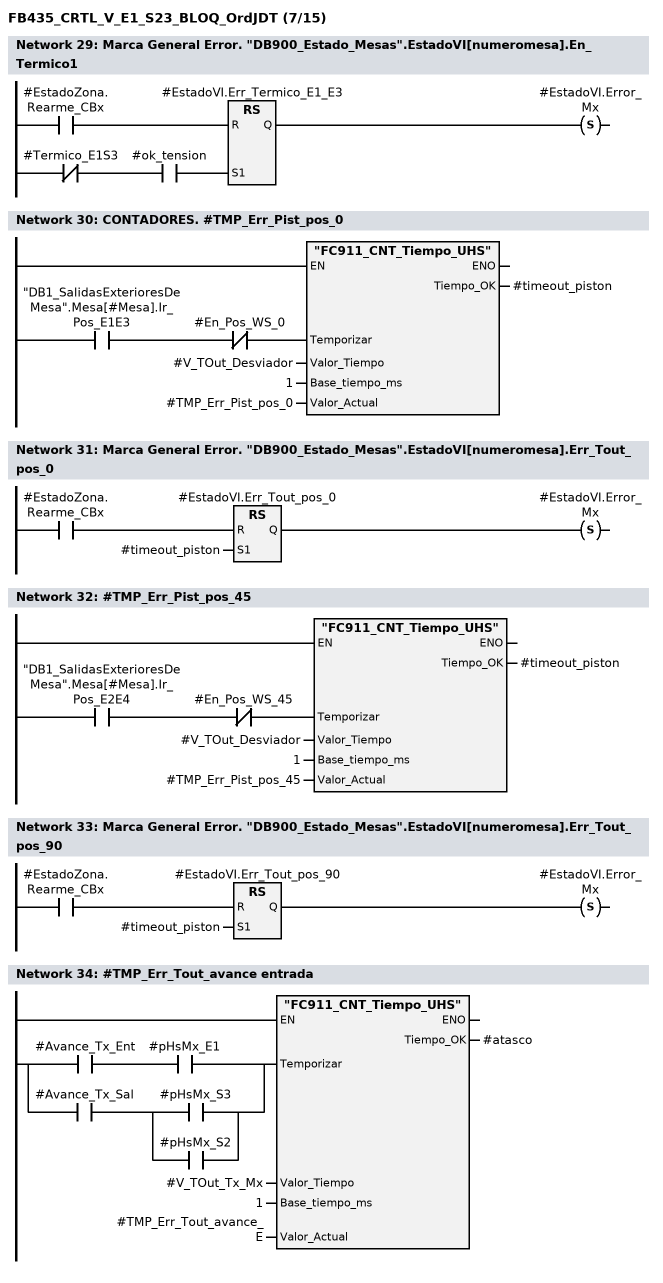
   RUNG wire#powerrail
      Contact( #EstadoZona.Rearme_CBx )
      S_RS(operand := #EstadoVI.Err_Termico_E1_E3, s1 := wire#w1)
      S_Coil( #EstadoVI.Error_Mx )
   END_RUNG
   RUNG wire#powerrail
      I_Contact( #Termico_E1S3 )
      Contact( #ok_tension )
   END_RUNG wire#w1
   // the same network as SCL:
   IF #EstadoZona.Rearme_CBx THEN
       #EstadoVI.Err_Termico_E1_E3 := FALSE;   // RS flip-flop
   END_IF;
   IF NOT #Termico_E1S3 AND #ok_tension THEN #EstadoVI.Err_Termico_E1_E3 := TRUE; END_IF;
   IF #EstadoVI.Err_Termico_E1_E3 THEN #EstadoVI.Error_Mx := TRUE; END_IF;
END_REGION

REGION Network 30: CONTADORES. #TMP_Err_Pist_pos_0
   RUNG wire#powerrail
      "FC911_CNT_Tiempo_UHS"(Temporizar := wire#w1, Valor_Tiempo := #V_TOut_Desviador, Base_tiempo_ms := 1, Valor_Actual := #TMP_Err_Pist_pos_0, Tiempo_OK => #timeout_piston)
   END_RUNG
   RUNG wire#powerrail
      Contact( "DB1_SalidasExterioresDeMesa".Mesa[#Mesa].Ir_Pos_E1E3 )
      I_Contact( #En_Pos_WS_0 )
   END_RUNG wire#w1
   // the same network as SCL:
   "FC911_CNT_Tiempo_UHS"(Temporizar := "DB1_SalidasExterioresDeMesa".Mesa[#Mesa].Ir_Pos_E1E3 AND NOT #En_Pos_WS_0,
                          Valor_Tiempo := #V_TOut_Desviador,
                          Base_tiempo_ms := 1,
                          Valor_Actual := #TMP_Err_Pist_pos_0,
                          Tiempo_OK => #timeout_piston);
END_REGION

REGION Network 31: Marca General Error. "DB900_Estado_Mesas".EstadoVI[numeromesa].Err_Tout_pos_0
   RUNG wire#powerrail
      Contact( #EstadoZona.Rearme_CBx )
      S_RS(operand := #EstadoVI.Err_Tout_pos_0, s1 := #timeout_piston)
      S_Coil( #EstadoVI.Error_Mx )
   END_RUNG
   // the same network as SCL:
   IF #EstadoZona.Rearme_CBx THEN
       #EstadoVI.Err_Tout_pos_0 := FALSE;   // RS flip-flop
   END_IF;
   IF #timeout_piston THEN #EstadoVI.Err_Tout_pos_0 := TRUE; END_IF;
   IF #EstadoVI.Err_Tout_pos_0 THEN #EstadoVI.Error_Mx := TRUE; END_IF;
END_REGION

REGION Network 32: #TMP_Err_Pist_pos_45
   RUNG wire#powerrail
      "FC911_CNT_Tiempo_UHS"(Temporizar := wire#w1, Valor_Tiempo := #V_TOut_Desviador, Base_tiempo_ms := 1, Valor_Actual := #TMP_Err_Pist_pos_45, Tiempo_OK => #timeout_piston)
   END_RUNG
   RUNG wire#powerrail
      Contact( "DB1_SalidasExterioresDeMesa".Mesa[#Mesa].Ir_Pos_E2E4 )
      I_Contact( #En_Pos_WS_45 )
   END_RUNG wire#w1
   // the same network as SCL:
   "FC911_CNT_Tiempo_UHS"(Temporizar := "DB1_SalidasExterioresDeMesa".Mesa[#Mesa].Ir_Pos_E2E4 AND NOT #En_Pos_WS_45,
                          Valor_Tiempo := #V_TOut_Desviador,
                          Base_tiempo_ms := 1,
                          Valor_Actual := #TMP_Err_Pist_pos_45,
                          Tiempo_OK => #timeout_piston);
END_REGION

REGION Network 33: Marca General Error. "DB900_Estado_Mesas".EstadoVI[numeromesa].Err_Tout_pos_90
   RUNG wire#powerrail
      Contact( #EstadoZona.Rearme_CBx )
      S_RS(operand := #EstadoVI.Err_Tout_pos_90, s1 := #timeout_piston)
      S_Coil( #EstadoVI.Error_Mx )
   END_RUNG
   // the same network as SCL:
   IF #EstadoZona.Rearme_CBx THEN
       #EstadoVI.Err_Tout_pos_90 := FALSE;   // RS flip-flop
   END_IF;
   IF #timeout_piston THEN #EstadoVI.Err_Tout_pos_90 := TRUE; END_IF;
   IF #EstadoVI.Err_Tout_pos_90 THEN #EstadoVI.Error_Mx := TRUE; END_IF;
END_REGION

REGION Network 34: #TMP_Err_Tout_avance entrada
   RUNG wire#powerrail
      "FC911_CNT_Tiempo_UHS"(Temporizar := wire#w2, Valor_Tiempo := #V_TOut_Tx_Mx, Base_tiempo_ms := 1, Valor_Actual := #TMP_Err_Tout_avance_E, Tiempo_OK => #atasco)
   END_RUNG
   RUNG wire#powerrail
      Contact( #Avance_Tx_Ent )
      Contact( #pHsMx_E1 )
   END_RUNG wire#w2
   RUNG wire#powerrail
      Contact( #Avance_Tx_Sal )
      wire#w1
      Contact( #pHsMx_S3 )
   END_RUNG wire#w2
   RUNG wire#w1
      Contact( #pHsMx_S2 )
   END_RUNG wire#w2
   // the same network as SCL:
   "FC911_CNT_Tiempo_UHS"(Temporizar := (#Avance_Tx_Ent AND #pHsMx_E1) OR (#Avance_Tx_Sal AND (#pHsMx_S3 OR #pHsMx_S2)),
                          Valor_Tiempo := #V_TOut_Tx_Mx,
                          Base_tiempo_ms := 1,
                          Valor_Actual := #TMP_Err_Tout_avance_E,
                          Tiempo_OK => #atasco);
END_REGION

REGION Network 35: Marca General Error. "DB900_Estado_Mesas".EstadoVI[numeromesa].Err_TOut_Avance_E1_E3
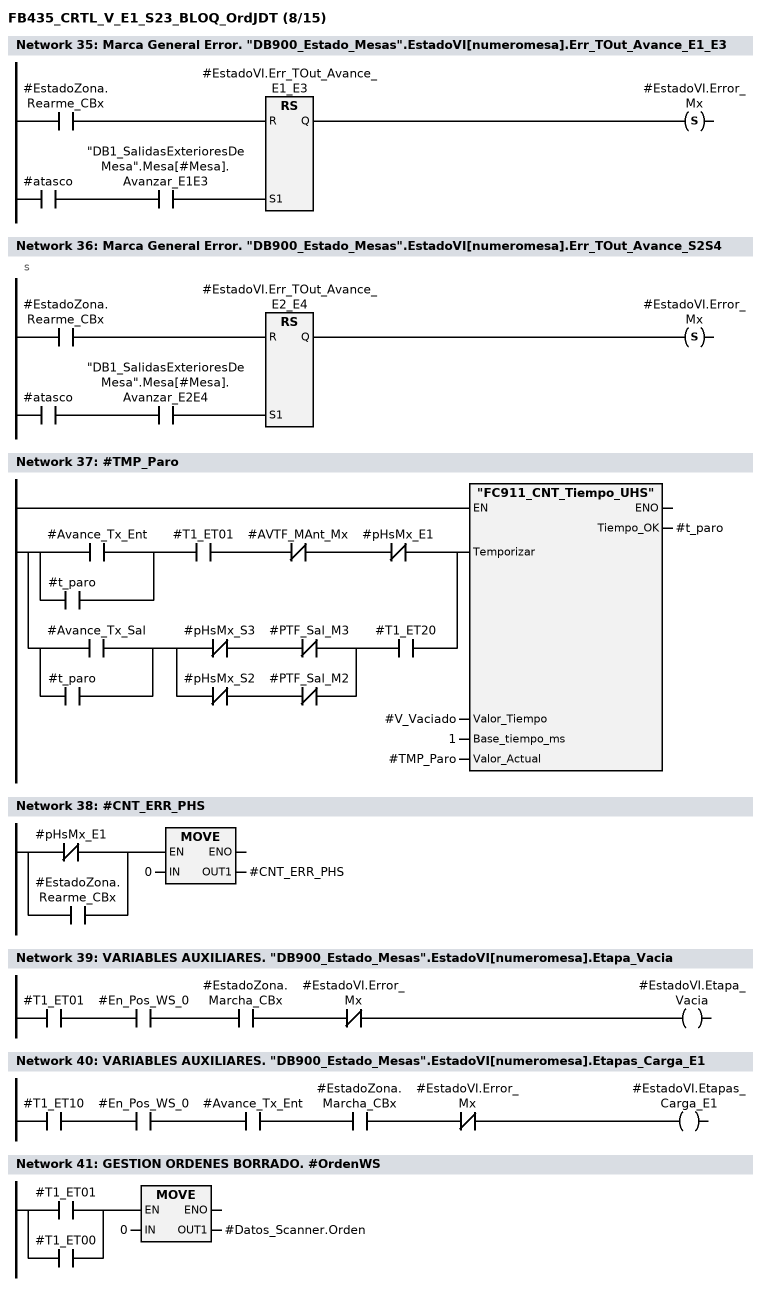
   RUNG wire#powerrail
      Contact( #EstadoZona.Rearme_CBx )
      S_RS(operand := #EstadoVI.Err_TOut_Avance_E1_E3, s1 := wire#w1)
      S_Coil( #EstadoVI.Error_Mx )
   END_RUNG
   RUNG wire#powerrail
      Contact( #atasco )
      Contact( "DB1_SalidasExterioresDeMesa".Mesa[#Mesa].Avanzar_E1E3 )
   END_RUNG wire#w1
   // the same network as SCL:
   IF #EstadoZona.Rearme_CBx THEN
       #EstadoVI.Err_TOut_Avance_E1_E3 := FALSE;   // RS flip-flop
   END_IF;
   IF #atasco AND "DB1_SalidasExterioresDeMesa".Mesa[#Mesa].Avanzar_E1E3 THEN
       #EstadoVI.Err_TOut_Avance_E1_E3 := TRUE;
   END_IF;
   IF #EstadoVI.Err_TOut_Avance_E1_E3 THEN #EstadoVI.Error_Mx := TRUE; END_IF;
END_REGION

REGION Network 36: Marca General Error. "DB900_Estado_Mesas".EstadoVI[numeromesa].Err_TOut_Avance_S2S4
   // s
   RUNG wire#powerrail
      Contact( #EstadoZona.Rearme_CBx )
      S_RS(operand := #EstadoVI.Err_TOut_Avance_E2_E4, s1 := wire#w1)
      S_Coil( #EstadoVI.Error_Mx )
   END_RUNG
   RUNG wire#powerrail
      Contact( #atasco )
      Contact( "DB1_SalidasExterioresDeMesa".Mesa[#Mesa].Avanzar_E2E4 )
   END_RUNG wire#w1
   // the same network as SCL:
   IF #EstadoZona.Rearme_CBx THEN
       #EstadoVI.Err_TOut_Avance_E2_E4 := FALSE;   // RS flip-flop
   END_IF;
   IF #atasco AND "DB1_SalidasExterioresDeMesa".Mesa[#Mesa].Avanzar_E2E4 THEN
       #EstadoVI.Err_TOut_Avance_E2_E4 := TRUE;
   END_IF;
   IF #EstadoVI.Err_TOut_Avance_E2_E4 THEN #EstadoVI.Error_Mx := TRUE; END_IF;
END_REGION

REGION Network 37: #TMP_Paro
   RUNG wire#powerrail
      "FC911_CNT_Tiempo_UHS"(Temporizar := wire#w4, Valor_Tiempo := #V_Vaciado, Base_tiempo_ms := 1, Valor_Actual := #TMP_Paro, Tiempo_OK => #t_paro)
   END_RUNG
   RUNG wire#powerrail
      Contact( #Avance_Tx_Ent )
      wire#w1
      Contact( #T1_ET01 )
      I_Contact( #AVTF_MAnt_Mx )
      I_Contact( #pHsMx_E1 )
   END_RUNG wire#w4
   RUNG wire#powerrail
      Contact( #t_paro )
   END_RUNG wire#w1
   RUNG wire#powerrail
      Contact( #Avance_Tx_Sal )
      wire#w2
      I_Contact( #pHsMx_S3 )
      I_Contact( #PTF_Sal_M3 )
      wire#w3
      Contact( #T1_ET20 )
   END_RUNG wire#w4
   RUNG wire#powerrail
      Contact( #t_paro )
   END_RUNG wire#w2
   RUNG wire#w2
      I_Contact( #pHsMx_S2 )
      I_Contact( #PTF_Sal_M2 )
   END_RUNG wire#w3
   // the same network as SCL:
   "FC911_CNT_Tiempo_UHS"(Temporizar := ((#Avance_Tx_Ent OR #t_paro) AND #T1_ET01 AND NOT #AVTF_MAnt_Mx AND NOT #pHsMx_E1) OR ((#Avance_Tx_Sal OR #t_paro) AND ((NOT #pHsMx_S3 AND NOT #PTF_Sal_M3) OR (NOT #pHsMx_S2 AND NOT #PTF_Sal_M2)) AND #T1_ET20),
                          Valor_Tiempo := #V_Vaciado,
                          Base_tiempo_ms := 1,
                          Valor_Actual := #TMP_Paro,
                          Tiempo_OK => #t_paro);
END_REGION

REGION Network 38: #CNT_ERR_PHS
   RUNG wire#powerrail
      I_Contact( #pHsMx_E1 )
      wire#w1
      { S7_GenerateENO := "TRUE" } Move(in := 0, out1 => #CNT_ERR_PHS)
   END_RUNG
   RUNG wire#powerrail
      Contact( #EstadoZona.Rearme_CBx )
   END_RUNG wire#w1
   // the same network as SCL:
   IF NOT #pHsMx_E1 OR #EstadoZona.Rearme_CBx THEN #CNT_ERR_PHS := 0; END_IF;
END_REGION

REGION Network 39: VARIABLES AUXILIARES. "DB900_Estado_Mesas".EstadoVI[numeromesa].Etapa_Vacia
   RUNG wire#powerrail
      Contact( #T1_ET01 )
      Contact( #En_Pos_WS_0 )
      Contact( #EstadoZona.Marcha_CBx )
      I_Contact( #EstadoVI.Error_Mx )
      Coil( #EstadoVI.Etapa_Vacia )
   END_RUNG
   // the same network as SCL:
   #EstadoVI.Etapa_Vacia := #T1_ET01 AND #En_Pos_WS_0 AND #EstadoZona.Marcha_CBx AND NOT #EstadoVI.Error_Mx;
END_REGION

REGION Network 40: VARIABLES AUXILIARES. "DB900_Estado_Mesas".EstadoVI[numeromesa].Etapas_Carga_E1
   RUNG wire#powerrail
      Contact( #T1_ET10 )
      Contact( #En_Pos_WS_0 )
      Contact( #Avance_Tx_Ent )
      Contact( #EstadoZona.Marcha_CBx )
      I_Contact( #EstadoVI.Error_Mx )
      Coil( #EstadoVI.Etapas_Carga_E1 )
   END_RUNG
   // the same network as SCL:
   #EstadoVI.Etapas_Carga_E1 := #T1_ET10 AND #En_Pos_WS_0 AND #Avance_Tx_Ent AND #EstadoZona.Marcha_CBx AND NOT #EstadoVI.Error_Mx;
END_REGION

REGION Network 41: GESTION ORDENES BORRADO. #OrdenWS
   RUNG wire#powerrail
      Contact( #T1_ET01 )
      wire#w1
      { S7_GenerateENO := "TRUE" } Move(in := 0, out1 => #Datos_Scanner.Orden)
   END_RUNG
   RUNG wire#powerrail
      Contact( #T1_ET00 )
   END_RUNG wire#w1
   // the same network as SCL:
   IF #T1_ET01 OR #T1_ET00 THEN #Datos_Scanner.Orden := 0; END_IF;
END_REGION

REGION Network 42: TOMA ORDENES FIFO. FC501
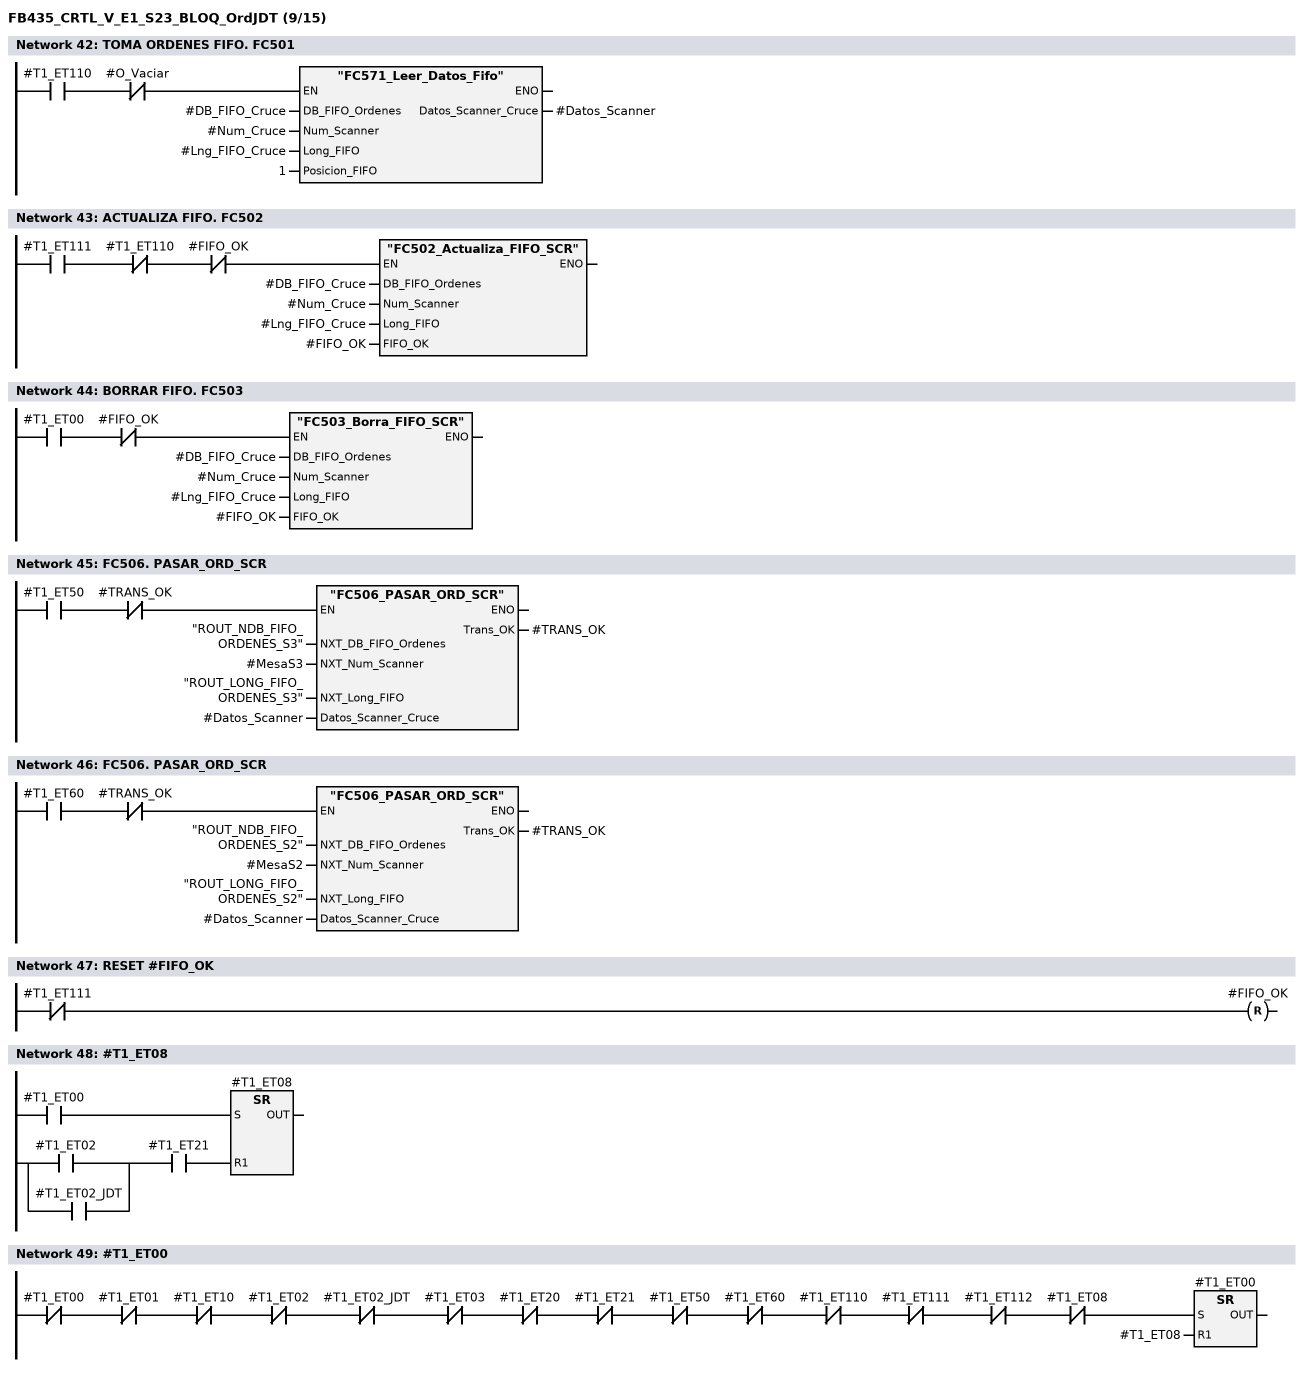
   RUNG wire#powerrail
      Contact( #T1_ET110 )
      I_Contact( #O_Vaciar )
      "FC571_Leer_Datos_Fifo"(DB_FIFO_Ordenes := #DB_FIFO_Cruce, Num_Scanner := #Num_Cruce, Long_FIFO := #Lng_FIFO_Cruce, Posicion_FIFO := 1, Datos_Scanner_Cruce => #Datos_Scanner)
   END_RUNG
   // the same network as SCL:
   IF #T1_ET110 AND NOT #O_Vaciar THEN
       "FC571_Leer_Datos_Fifo"(DB_FIFO_Ordenes := #DB_FIFO_Cruce,
                               Num_Scanner := #Num_Cruce,
                               Long_FIFO := #Lng_FIFO_Cruce,
                               Posicion_FIFO := 1,
                               Datos_Scanner_Cruce => #Datos_Scanner);
   END_IF;
END_REGION

REGION Network 43: ACTUALIZA FIFO. FC502
   RUNG wire#powerrail
      Contact( #T1_ET111 )
      I_Contact( #T1_ET110 )
      I_Contact( #FIFO_OK )
      "FC502_Actualiza_FIFO_SCR"(DB_FIFO_Ordenes := #DB_FIFO_Cruce, Num_Scanner := #Num_Cruce, Long_FIFO := #Lng_FIFO_Cruce, FIFO_OK := #FIFO_OK)
   END_RUNG
   // the same network as SCL:
   IF #T1_ET111 AND NOT #T1_ET110 AND NOT #FIFO_OK THEN
       "FC502_Actualiza_FIFO_SCR"(DB_FIFO_Ordenes := #DB_FIFO_Cruce,
                               Num_Scanner := #Num_Cruce,
                               Long_FIFO := #Lng_FIFO_Cruce,
                               FIFO_OK := #FIFO_OK);
   END_IF;
END_REGION

REGION Network 44: BORRAR FIFO. FC503
   RUNG wire#powerrail
      Contact( #T1_ET00 )
      I_Contact( #FIFO_OK )
      "FC503_Borra_FIFO_SCR"(DB_FIFO_Ordenes := #DB_FIFO_Cruce, Num_Scanner := #Num_Cruce, Long_FIFO := #Lng_FIFO_Cruce, FIFO_OK := #FIFO_OK)
   END_RUNG
   // the same network as SCL:
   IF #T1_ET00 AND NOT #FIFO_OK THEN
       "FC503_Borra_FIFO_SCR"(DB_FIFO_Ordenes := #DB_FIFO_Cruce,
                              Num_Scanner := #Num_Cruce,
                              Long_FIFO := #Lng_FIFO_Cruce,
                              FIFO_OK := #FIFO_OK);
   END_IF;
END_REGION

REGION Network 45: FC506. PASAR_ORD_SCR
   RUNG wire#powerrail
      Contact( #T1_ET50 )
      I_Contact( #TRANS_OK )
      "FC506_PASAR_ORD_SCR"(NXT_DB_FIFO_Ordenes := "ROUT_NDB_FIFO_ORDENES_S3", NXT_Num_Scanner := #MesaS3, NXT_Long_FIFO := "ROUT_LONG_FIFO_ORDENES_S3", Datos_Scanner_Cruce := #Datos_Scanner, Trans_OK => #TRANS_OK)
   END_RUNG
   // the same network as SCL:
   IF #T1_ET50 AND NOT #TRANS_OK THEN
       "FC506_PASAR_ORD_SCR"(NXT_DB_FIFO_Ordenes := "ROUT_NDB_FIFO_ORDENES_S3",
                             NXT_Num_Scanner := #MesaS3,
                             NXT_Long_FIFO := "ROUT_LONG_FIFO_ORDENES_S3",
                             Datos_Scanner_Cruce := #Datos_Scanner,
                             Trans_OK => #TRANS_OK);
   END_IF;
END_REGION

REGION Network 46: FC506. PASAR_ORD_SCR
   RUNG wire#powerrail
      Contact( #T1_ET60 )
      I_Contact( #TRANS_OK )
      "FC506_PASAR_ORD_SCR"(NXT_DB_FIFO_Ordenes := "ROUT_NDB_FIFO_ORDENES_S2", NXT_Num_Scanner := #MesaS2, NXT_Long_FIFO := "ROUT_LONG_FIFO_ORDENES_S2", Datos_Scanner_Cruce := #Datos_Scanner, Trans_OK => #TRANS_OK)
   END_RUNG
   // the same network as SCL:
   IF #T1_ET60 AND NOT #TRANS_OK THEN
       "FC506_PASAR_ORD_SCR"(NXT_DB_FIFO_Ordenes := "ROUT_NDB_FIFO_ORDENES_S2",
                             NXT_Num_Scanner := #MesaS2,
                             NXT_Long_FIFO := "ROUT_LONG_FIFO_ORDENES_S2",
                             Datos_Scanner_Cruce := #Datos_Scanner,
                             Trans_OK => #TRANS_OK);
   END_IF;
END_REGION

REGION Network 47: RESET #FIFO_OK
   RUNG wire#powerrail
      I_Contact( #T1_ET111 )
      R_Coil( #FIFO_OK )
   END_RUNG
   // the same network as SCL:
   IF NOT #T1_ET111 THEN #FIFO_OK := FALSE; END_IF;
END_REGION

REGION Network 48: #T1_ET08
   RUNG wire#powerrail
      Contact( #T1_ET00 )
      S_SR(operand := #T1_ET08, r1 := wire#w2)
   END_RUNG
   RUNG wire#powerrail
      Contact( #T1_ET02 )
      wire#w1
      Contact( #T1_ET21 )
   END_RUNG wire#w2
   RUNG wire#powerrail
      Contact( #T1_ET02_JDT )
   END_RUNG wire#w1
   // the same network as SCL:
   IF #T1_ET00 THEN
       #T1_ET08 := TRUE;   // SR flip-flop
   END_IF;
   IF (#T1_ET02 OR #T1_ET02_JDT) AND #T1_ET21 THEN #T1_ET08 := FALSE; END_IF;
END_REGION

REGION Network 49: #T1_ET00
   RUNG wire#powerrail
      I_Contact( #T1_ET00 )
      I_Contact( #T1_ET01 )
      I_Contact( #T1_ET10 )
      I_Contact( #T1_ET02 )
      I_Contact( #T1_ET02_JDT )
      I_Contact( #T1_ET03 )
      I_Contact( #T1_ET20 )
      I_Contact( #T1_ET21 )
      I_Contact( #T1_ET50 )
      I_Contact( #T1_ET60 )
      I_Contact( #T1_ET110 )
      I_Contact( #T1_ET111 )
      I_Contact( #T1_ET112 )
      I_Contact( #T1_ET08 )
      S_SR(operand := #T1_ET00, r1 := #T1_ET08)
   END_RUNG
   // the same network as SCL:
   IF NOT #T1_ET00 AND NOT #T1_ET01 AND NOT #T1_ET10 AND NOT #T1_ET02 AND NOT #T1_ET02_JDT AND NOT #T1_ET03 AND NOT #T1_ET20 AND NOT #T1_ET21 AND NOT #T1_ET50 AND NOT #T1_ET60 AND NOT #T1_ET110 AND NOT #T1_ET111 AND NOT #T1_ET112 AND NOT #T1_ET08 THEN
       #T1_ET00 := TRUE;   // SR flip-flop
   END_IF;
   IF #T1_ET08 THEN #T1_ET00 := FALSE; END_IF;
END_REGION

REGION Network 50: RESET #TRANS_OK
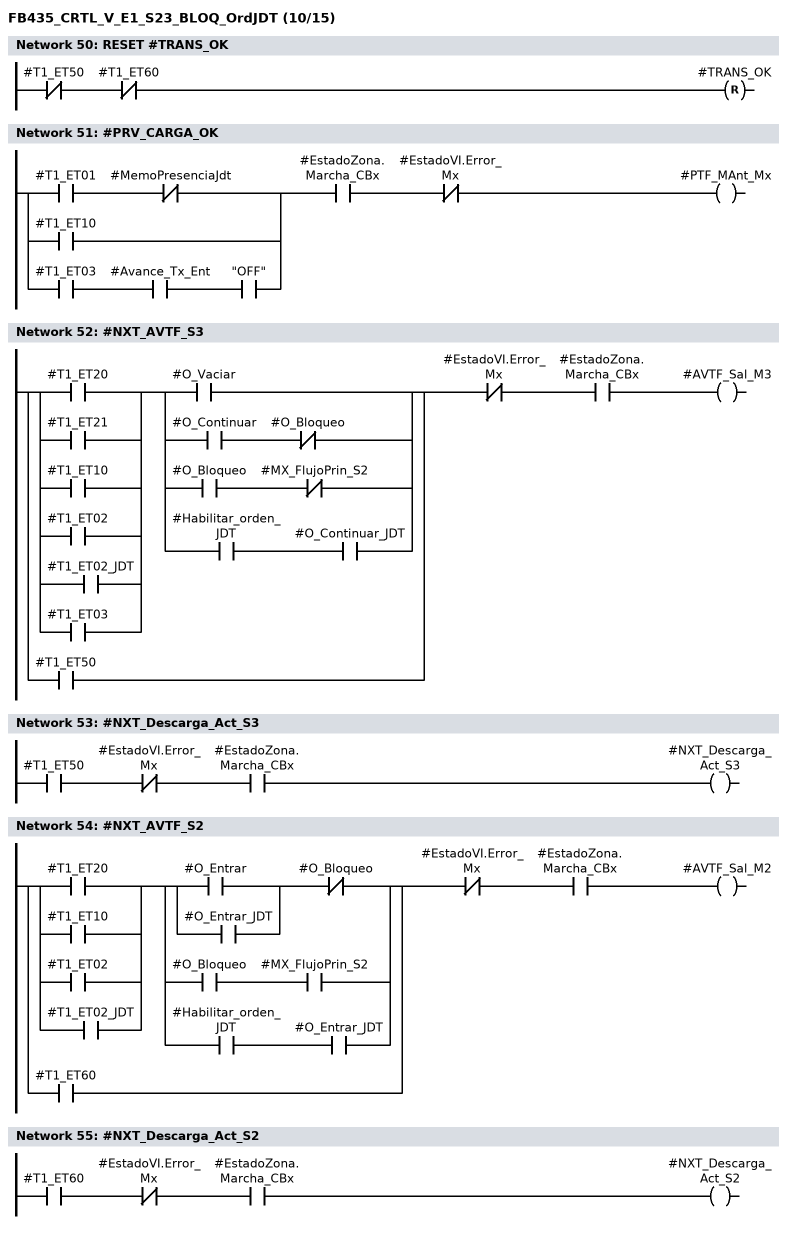
   RUNG wire#powerrail
      I_Contact( #T1_ET50 )
      I_Contact( #T1_ET60 )
      R_Coil( #TRANS_OK )
   END_RUNG
   // the same network as SCL:
   IF NOT #T1_ET50 AND NOT #T1_ET60 THEN #TRANS_OK := FALSE; END_IF;
END_REGION

REGION Network 51: #PRV_CARGA_OK
   RUNG wire#powerrail
      Contact( #T1_ET01 )
      I_Contact( #MemoPresenciaJdt )
      wire#w1
      Contact( #EstadoZona.Marcha_CBx )
      I_Contact( #EstadoVI.Error_Mx )
      Coil( #PTF_MAnt_Mx )
   END_RUNG
   RUNG wire#powerrail
      Contact( #T1_ET10 )
   END_RUNG wire#w1
   RUNG wire#powerrail
      Contact( #T1_ET03 )
      Contact( #Avance_Tx_Ent )
      Contact( "OFF" )
   END_RUNG wire#w1
   // the same network as SCL:
   #PTF_MAnt_Mx := ((#T1_ET01 AND NOT #MemoPresenciaJdt) OR #T1_ET10 OR (#T1_ET03 AND #Avance_Tx_Ent AND "OFF")) AND #EstadoZona.Marcha_CBx AND NOT #EstadoVI.Error_Mx;
END_REGION

REGION Network 52: #NXT_AVTF_S3
   RUNG wire#powerrail
      Contact( #T1_ET20 )
      wire#w1
      Contact( #O_Vaciar )
      wire#w2
      I_Contact( #EstadoVI.Error_Mx )
      Contact( #EstadoZona.Marcha_CBx )
      Coil( #AVTF_Sal_M3 )
   END_RUNG
   RUNG wire#powerrail
      Contact( #T1_ET21 )
   END_RUNG wire#w1
   RUNG wire#powerrail
      Contact( #T1_ET10 )
   END_RUNG wire#w1
   RUNG wire#powerrail
      Contact( #T1_ET02 )
   END_RUNG wire#w1
   RUNG wire#powerrail
      Contact( #T1_ET02_JDT )
   END_RUNG wire#w1
   RUNG wire#powerrail
      Contact( #T1_ET03 )
   END_RUNG wire#w1
   RUNG wire#w1
      Contact( #O_Continuar )
      I_Contact( #O_Bloqueo )
   END_RUNG wire#w2
   RUNG wire#w1
      Contact( #O_Bloqueo )
      I_Contact( #MX_FlujoPrin_S2 )
   END_RUNG wire#w2
   RUNG wire#w1
      Contact( #Habilitar_orden_JDT )
      Contact( #O_Continuar_JDT )
   END_RUNG wire#w2
   RUNG wire#powerrail
      Contact( #T1_ET50 )
   END_RUNG wire#w2
   // the same network as SCL:
   #AVTF_Sal_M3 := (((#T1_ET20 OR #T1_ET21 OR #T1_ET10 OR #T1_ET02 OR #T1_ET02_JDT OR #T1_ET03) AND (#O_Vaciar OR (#O_Continuar AND NOT #O_Bloqueo) OR (#O_Bloqueo AND NOT #MX_FlujoPrin_S2) OR (#Habilitar_orden_JDT AND #O_Continuar_JDT))) OR #T1_ET50) AND NOT #EstadoVI.Error_Mx AND #EstadoZona.Marcha_CBx;
END_REGION

REGION Network 53: #NXT_Descarga_Act_S3
   RUNG wire#powerrail
      Contact( #T1_ET50 )
      I_Contact( #EstadoVI.Error_Mx )
      Contact( #EstadoZona.Marcha_CBx )
      Coil( #NXT_Descarga_Act_S3 )
   END_RUNG
   // the same network as SCL:
   #NXT_Descarga_Act_S3 := #T1_ET50 AND NOT #EstadoVI.Error_Mx AND #EstadoZona.Marcha_CBx;
END_REGION

REGION Network 54: #NXT_AVTF_S2
   RUNG wire#powerrail
      Contact( #T1_ET20 )
      wire#w1
      Contact( #O_Entrar )
      wire#w2
      I_Contact( #O_Bloqueo )
      wire#w3
      I_Contact( #EstadoVI.Error_Mx )
      Contact( #EstadoZona.Marcha_CBx )
      Coil( #AVTF_Sal_M2 )
   END_RUNG
   RUNG wire#powerrail
      Contact( #T1_ET10 )
   END_RUNG wire#w1
   RUNG wire#powerrail
      Contact( #T1_ET02 )
   END_RUNG wire#w1
   RUNG wire#powerrail
      Contact( #T1_ET02_JDT )
   END_RUNG wire#w1
   RUNG wire#w1
      Contact( #O_Entrar_JDT )
   END_RUNG wire#w2
   RUNG wire#w1
      Contact( #O_Bloqueo )
      Contact( #MX_FlujoPrin_S2 )
   END_RUNG wire#w3
   RUNG wire#w1
      Contact( #Habilitar_orden_JDT )
      Contact( #O_Entrar_JDT )
   END_RUNG wire#w3
   RUNG wire#powerrail
      Contact( #T1_ET60 )
   END_RUNG wire#w3
   // the same network as SCL:
   #AVTF_Sal_M2 := (((#T1_ET20 OR #T1_ET10 OR #T1_ET02 OR #T1_ET02_JDT) AND (((#O_Entrar OR #O_Entrar_JDT) AND NOT #O_Bloqueo) OR (#O_Bloqueo AND #MX_FlujoPrin_S2) OR (#Habilitar_orden_JDT AND #O_Entrar_JDT))) OR #T1_ET60) AND NOT #EstadoVI.Error_Mx AND #EstadoZona.Marcha_CBx;
END_REGION

REGION Network 55: #NXT_Descarga_Act_S2
   RUNG wire#powerrail
      Contact( #T1_ET60 )
      I_Contact( #EstadoVI.Error_Mx )
      Contact( #EstadoZona.Marcha_CBx )
      Coil( #NXT_Descarga_Act_S2 )
   END_RUNG
   // the same network as SCL:
   #NXT_Descarga_Act_S2 := #T1_ET60 AND NOT #EstadoVI.Error_Mx AND #EstadoZona.Marcha_CBx;
END_REGION

REGION Network 56: #MA_IR_POS_S2
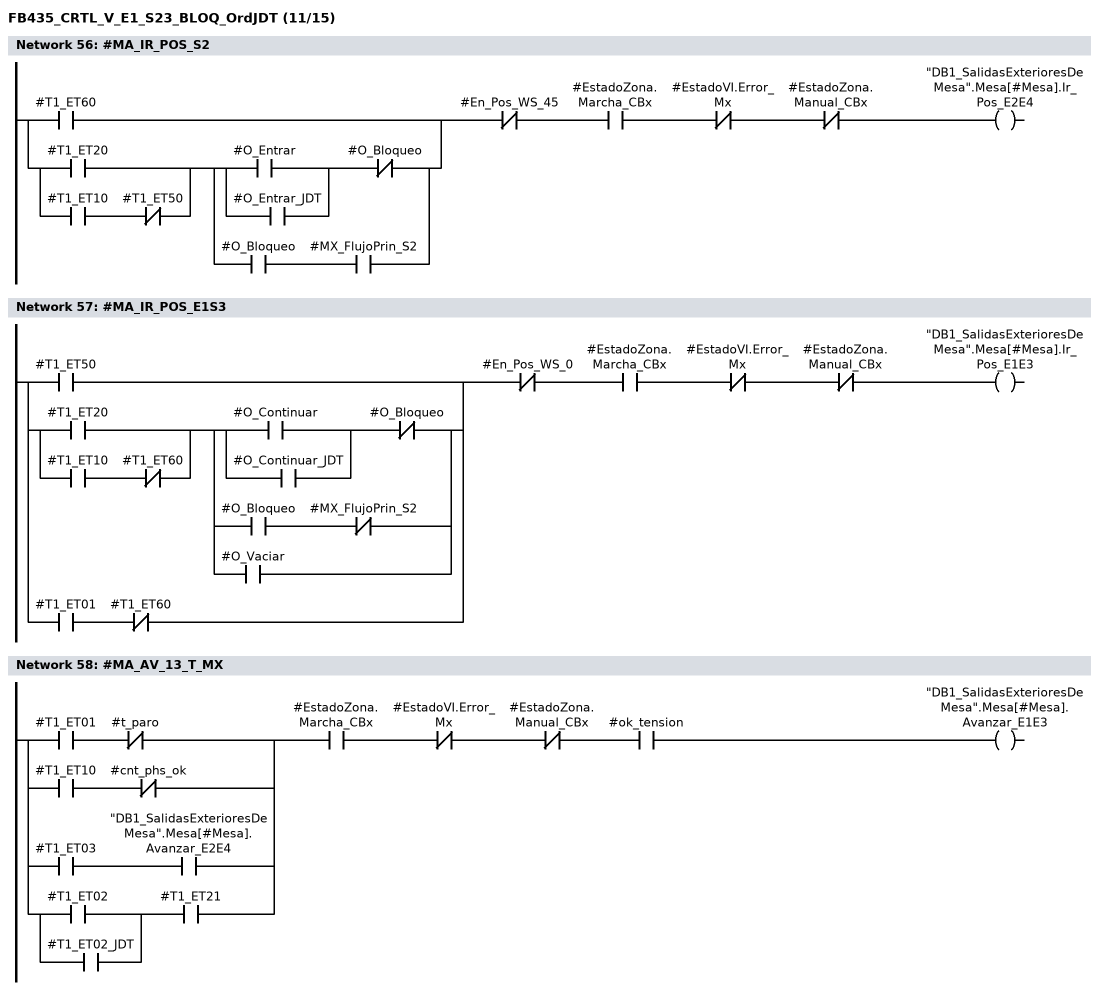
   RUNG wire#powerrail
      Contact( #T1_ET60 )
      wire#w1
      I_Contact( #En_Pos_WS_45 )
      Contact( #EstadoZona.Marcha_CBx )
      I_Contact( #EstadoVI.Error_Mx )
      I_Contact( #EstadoZona.Manual_CBx )
      Coil( "DB1_SalidasExterioresDeMesa".Mesa[#Mesa].Ir_Pos_E2E4 )
   END_RUNG
   RUNG wire#powerrail
      Contact( #T1_ET20 )
      wire#w2
      Contact( #O_Entrar )
      wire#w3
      I_Contact( #O_Bloqueo )
   END_RUNG wire#w1
   RUNG wire#powerrail
      Contact( #T1_ET10 )
      I_Contact( #T1_ET50 )
   END_RUNG wire#w2
   RUNG wire#w2
      Contact( #O_Entrar_JDT )
   END_RUNG wire#w3
   RUNG wire#w2
      Contact( #O_Bloqueo )
      Contact( #MX_FlujoPrin_S2 )
   END_RUNG wire#w1
   // the same network as SCL:
   "DB1_SalidasExterioresDeMesa".Mesa[#Mesa].Ir_Pos_E2E4 := (#T1_ET60 OR ((#T1_ET20 OR (#T1_ET10 AND NOT #T1_ET50)) AND (((#O_Entrar OR #O_Entrar_JDT) AND NOT #O_Bloqueo) OR (#O_Bloqueo AND #MX_FlujoPrin_S2)))) AND NOT #En_Pos_WS_45 AND #EstadoZona.Marcha_CBx AND NOT #EstadoVI.Error_Mx AND NOT #EstadoZona.Manual_CBx;
END_REGION

REGION Network 57: #MA_IR_POS_E1S3
   RUNG wire#powerrail
      Contact( #T1_ET50 )
      wire#w1
      I_Contact( #En_Pos_WS_0 )
      Contact( #EstadoZona.Marcha_CBx )
      I_Contact( #EstadoVI.Error_Mx )
      I_Contact( #EstadoZona.Manual_CBx )
      Coil( "DB1_SalidasExterioresDeMesa".Mesa[#Mesa].Ir_Pos_E1E3 )
   END_RUNG
   RUNG wire#powerrail
      Contact( #T1_ET20 )
      wire#w2
      Contact( #O_Continuar )
      wire#w3
      I_Contact( #O_Bloqueo )
   END_RUNG wire#w1
   RUNG wire#powerrail
      Contact( #T1_ET10 )
      I_Contact( #T1_ET60 )
   END_RUNG wire#w2
   RUNG wire#w2
      Contact( #O_Continuar_JDT )
   END_RUNG wire#w3
   RUNG wire#w2
      Contact( #O_Bloqueo )
      I_Contact( #MX_FlujoPrin_S2 )
   END_RUNG wire#w1
   RUNG wire#w2
      Contact( #O_Vaciar )
   END_RUNG wire#w1
   RUNG wire#powerrail
      Contact( #T1_ET01 )
      I_Contact( #T1_ET60 )
   END_RUNG wire#w1
   // the same network as SCL:
   "DB1_SalidasExterioresDeMesa".Mesa[#Mesa].Ir_Pos_E1E3 := (#T1_ET50 OR ((#T1_ET20 OR (#T1_ET10 AND NOT #T1_ET60)) AND (((#O_Continuar OR #O_Continuar_JDT) AND NOT #O_Bloqueo) OR (#O_Bloqueo AND NOT #MX_FlujoPrin_S2) OR #O_Vaciar)) OR (#T1_ET01 AND NOT #T1_ET60)) AND NOT #En_Pos_WS_0 AND #EstadoZona.Marcha_CBx AND NOT #EstadoVI.Error_Mx AND NOT #EstadoZona.Manual_CBx;
END_REGION

REGION Network 58: #MA_AV_13_T_MX
   RUNG wire#powerrail
      Contact( #T1_ET01 )
      I_Contact( #t_paro )
      wire#w1
      Contact( #EstadoZona.Marcha_CBx )
      I_Contact( #EstadoVI.Error_Mx )
      I_Contact( #EstadoZona.Manual_CBx )
      Contact( #ok_tension )
      Coil( "DB1_SalidasExterioresDeMesa".Mesa[#Mesa].Avanzar_E1E3 )
   END_RUNG
   RUNG wire#powerrail
      Contact( #T1_ET10 )
      I_Contact( #cnt_phs_ok )
   END_RUNG wire#w1
   RUNG wire#powerrail
      Contact( #T1_ET03 )
      Contact( "DB1_SalidasExterioresDeMesa".Mesa[#Mesa].Avanzar_E2E4 )
   END_RUNG wire#w1
   RUNG wire#powerrail
      Contact( #T1_ET02 )
      wire#w2
      Contact( #T1_ET21 )
   END_RUNG wire#w1
   RUNG wire#powerrail
      Contact( #T1_ET02_JDT )
   END_RUNG wire#w2
   // the same network as SCL:
   "DB1_SalidasExterioresDeMesa".Mesa[#Mesa].Avanzar_E1E3 := ((#T1_ET01 AND NOT #t_paro) OR (#T1_ET10 AND NOT #cnt_phs_ok) OR (#T1_ET03 AND "DB1_SalidasExterioresDeMesa".Mesa[#Mesa].Avanzar_E2E4) OR ((#T1_ET02 OR #T1_ET02_JDT) AND #T1_ET21)) AND #EstadoZona.Marcha_CBx AND NOT #EstadoVI.Error_Mx AND NOT #EstadoZona.Manual_CBx AND #ok_tension;
END_REGION

REGION Network 59: #MA_AV_24_TR_MX
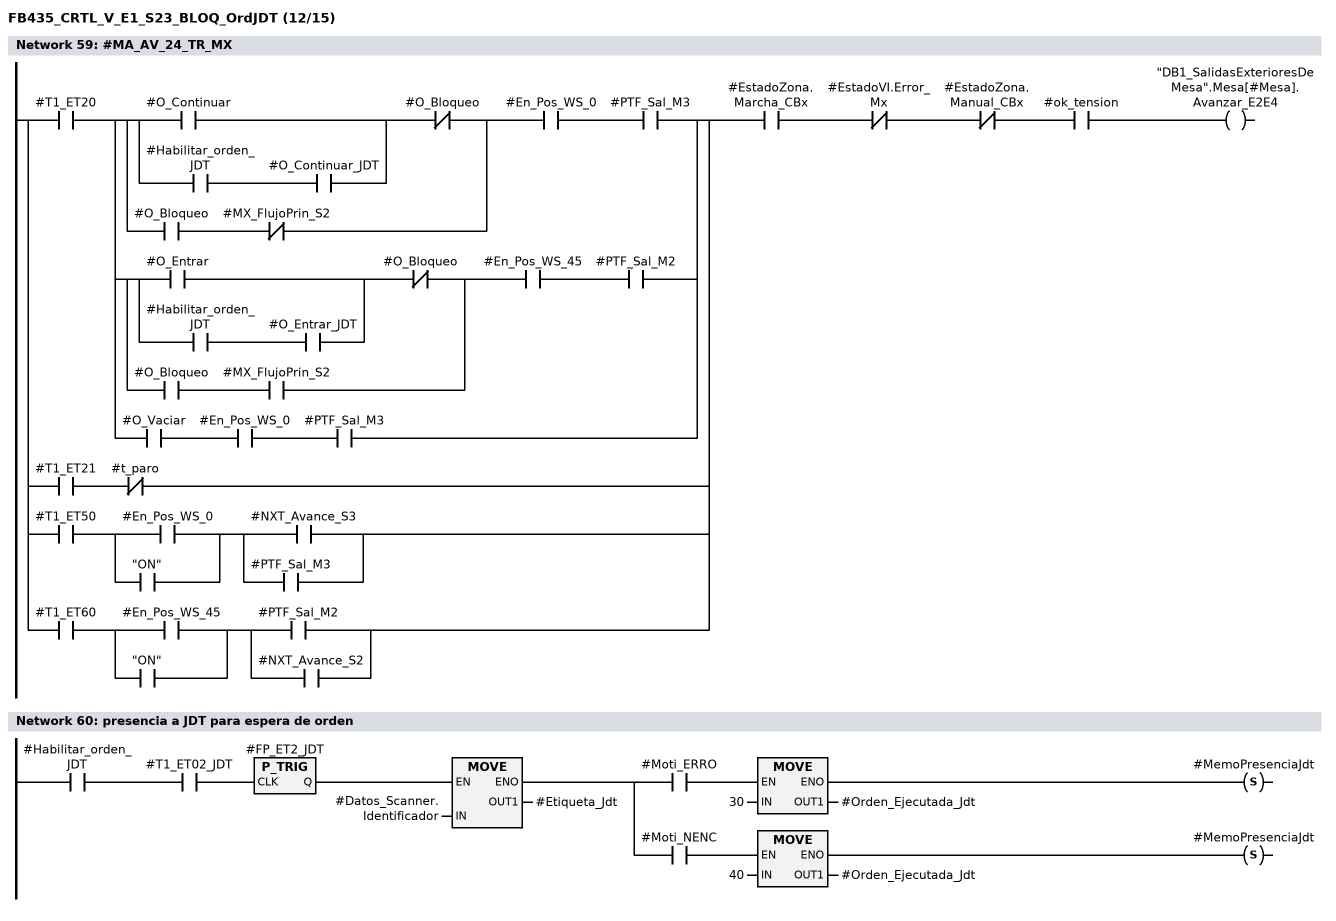
   RUNG wire#powerrail
      Contact( #T1_ET20 )
      wire#w1
      Contact( #O_Continuar )
      wire#w2
      I_Contact( #O_Bloqueo )
      wire#w3
      Contact( #En_Pos_WS_0 )
      Contact( #PTF_Sal_M3 )
      wire#w4
      Contact( #EstadoZona.Marcha_CBx )
      I_Contact( #EstadoVI.Error_Mx )
      I_Contact( #EstadoZona.Manual_CBx )
      Contact( #ok_tension )
      Coil( "DB1_SalidasExterioresDeMesa".Mesa[#Mesa].Avanzar_E2E4 )
   END_RUNG
   RUNG wire#w1
      Contact( #Habilitar_orden_JDT )
      Contact( #O_Continuar_JDT )
   END_RUNG wire#w2
   RUNG wire#w1
      Contact( #O_Bloqueo )
      I_Contact( #MX_FlujoPrin_S2 )
   END_RUNG wire#w3
   RUNG wire#w1
      Contact( #O_Entrar )
      wire#w5
      I_Contact( #O_Bloqueo )
      wire#w6
      Contact( #En_Pos_WS_45 )
      Contact( #PTF_Sal_M2 )
   END_RUNG wire#w4
   RUNG wire#w1
      Contact( #Habilitar_orden_JDT )
      Contact( #O_Entrar_JDT )
   END_RUNG wire#w5
   RUNG wire#w1
      Contact( #O_Bloqueo )
      Contact( #MX_FlujoPrin_S2 )
   END_RUNG wire#w6
   RUNG wire#w1
      Contact( #O_Vaciar )
      Contact( #En_Pos_WS_0 )
      Contact( #PTF_Sal_M3 )
   END_RUNG wire#w4
   RUNG wire#powerrail
      Contact( #T1_ET21 )
      I_Contact( #t_paro )
   END_RUNG wire#w4
   RUNG wire#powerrail
      Contact( #T1_ET50 )
      wire#w7
      Contact( #En_Pos_WS_0 )
      wire#w8
      Contact( #NXT_Avance_S3 )
   END_RUNG wire#w4
   RUNG wire#w7
      Contact( "ON" )
   END_RUNG wire#w8
   RUNG wire#w8
      Contact( #PTF_Sal_M3 )
   END_RUNG wire#w4
   RUNG wire#powerrail
      Contact( #T1_ET60 )
      wire#w9
      Contact( #En_Pos_WS_45 )
      wire#w10
      Contact( #PTF_Sal_M2 )
   END_RUNG wire#w4
   RUNG wire#w9
      Contact( "ON" )
   END_RUNG wire#w10
   RUNG wire#w10
      Contact( #NXT_Avance_S2 )
   END_RUNG wire#w4
   // the same network as SCL:
   "DB1_SalidasExterioresDeMesa".Mesa[#Mesa].Avanzar_E2E4 := ((#T1_ET20 AND (((((#O_Continuar OR (#Habilitar_orden_JDT AND #O_Continuar_JDT)) AND NOT #O_Bloqueo) OR (#O_Bloqueo AND NOT #MX_FlujoPrin_S2)) AND #En_Pos_WS_0 AND #PTF_Sal_M3) OR ((((#O_Entrar OR (#Habilitar_orden_JDT AND #O_Entrar_JDT)) AND NOT #O_Bloqueo) OR (#O_Bloqueo AND #MX_FlujoPrin_S2)) AND #En_Pos_WS_45 AND #PTF_Sal_M2) OR (#O_Vaciar AND #En_Pos_WS_0 AND #PTF_Sal_M3))) OR (#T1_ET21 AND NOT #t_paro) OR (#T1_ET50 AND (#En_Pos_WS_0 OR "ON") AND (#NXT_Avance_S3 OR #PTF_Sal_M3)) OR (#T1_ET60 AND (#En_Pos_WS_45 OR "ON") AND (#PTF_Sal_M2 OR #NXT_Avance_S2))) AND #EstadoZona.Marcha_CBx AND NOT #EstadoVI.Error_Mx AND NOT #EstadoZona.Manual_CBx AND #ok_tension;
END_REGION

REGION Network 60: presencia a JDT para espera de orden
   RUNG wire#powerrail
      Contact( #Habilitar_orden_JDT )
      Contact( #T1_ET02_JDT )
      P_Trig( #FP_ET2_JDT )
      { S7_GenerateENO := "TRUE" } Move(in := #Datos_Scanner.Identificador, out1 => #Etiqueta_Jdt)
      wire#w1
      Contact( #Moti_ERRO )
      { S7_GenerateENO := "TRUE" } Move(in := 30, out1 => #Orden_Ejecutada_Jdt)
      S_Coil( #MemoPresenciaJdt )
   END_RUNG
   RUNG wire#w1
      Contact( #Moti_NENC )
      { S7_GenerateENO := "TRUE" } Move(in := 40, out1 => #Orden_Ejecutada_Jdt)
      S_Coil( #MemoPresenciaJdt )
   END_RUNG
   // the same network as SCL:
   // ENO of a box is taken as its EN; it also drops when the box reports an error
   #_w1 := #Habilitar_orden_JDT AND #T1_ET02_JDT;
   #_w2 := #_w1 AND NOT #FP_ET2_JDT;   // rising edge
   #FP_ET2_JDT := #_w1;
   IF #_w2 THEN #Etiqueta_Jdt := #Datos_Scanner.Identificador; END_IF;
   IF #_w2 AND #Moti_ERRO THEN
       #Orden_Ejecutada_Jdt := 30;
       #MemoPresenciaJdt := TRUE;
   END_IF;
   IF #_w2 AND #Moti_NENC THEN
       #Orden_Ejecutada_Jdt := 40;
       #MemoPresenciaJdt := TRUE;
   END_IF;
END_REGION

REGION Network 61: PASAR ETIQUETA JDT
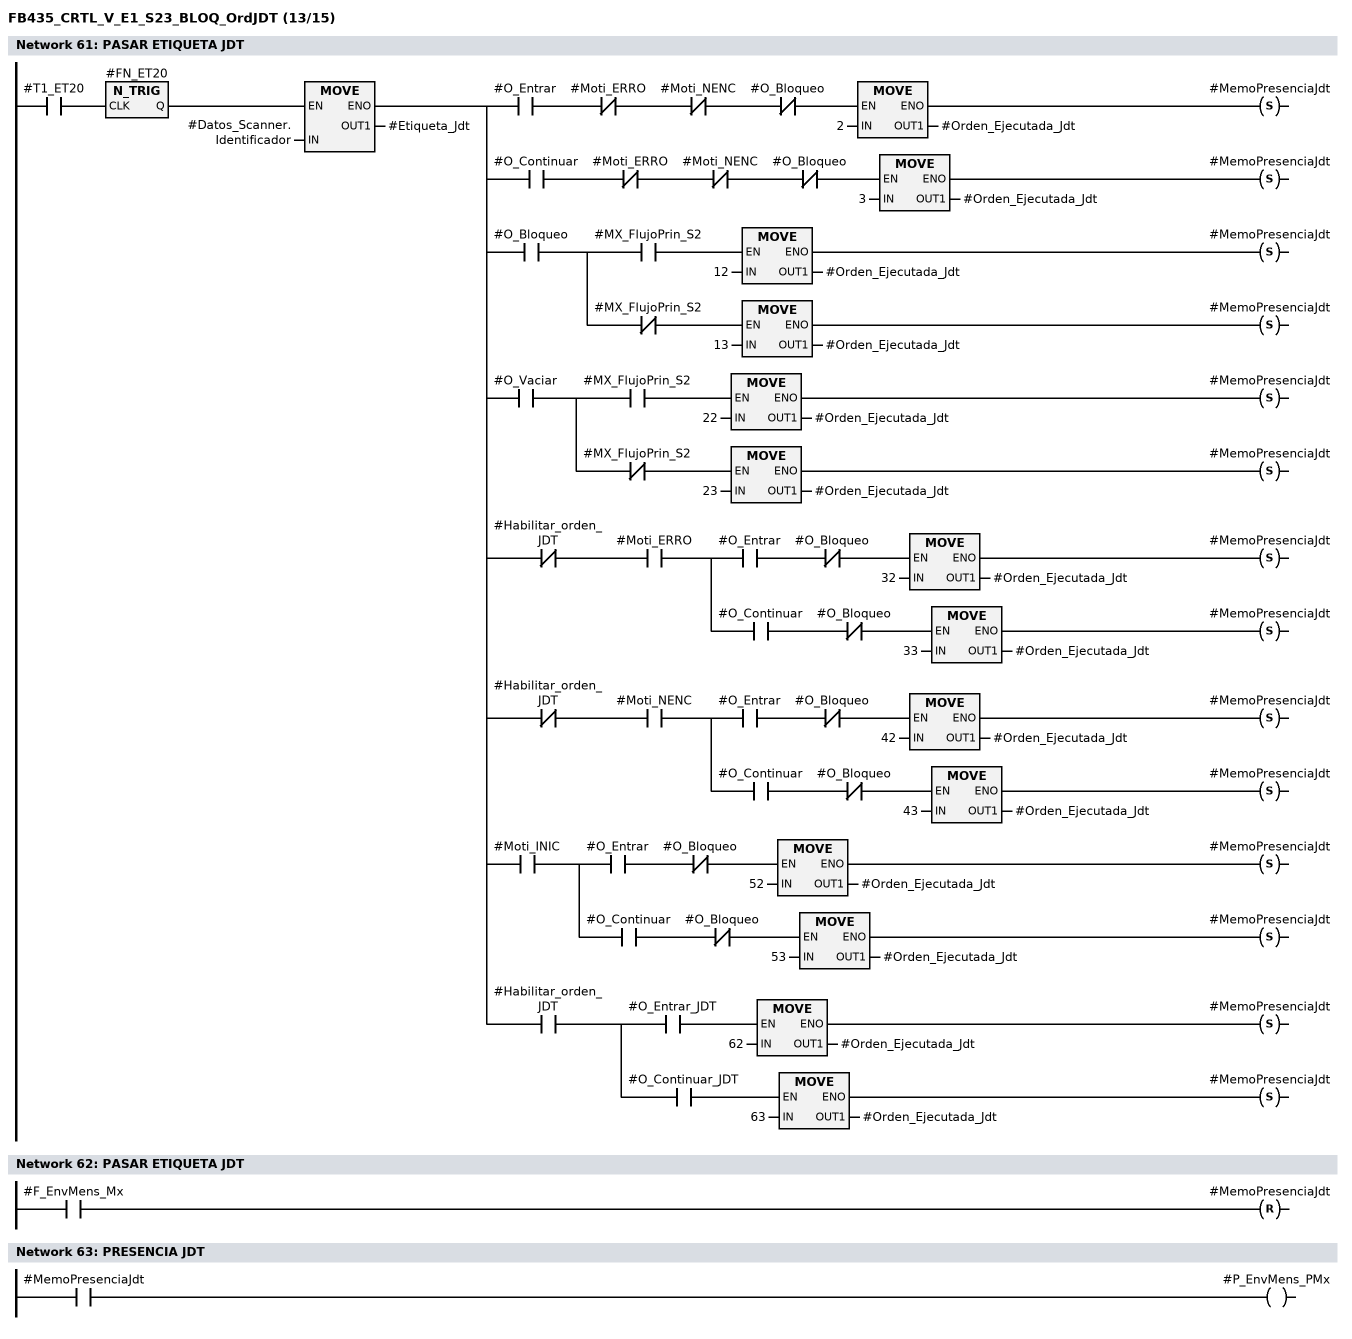
   RUNG wire#powerrail
      Contact( #T1_ET20 )
      N_Trig( #FN_ET20 )
      { S7_GenerateENO := "TRUE" } Move(in := #Datos_Scanner.Identificador, out1 => #Etiqueta_Jdt)
      wire#w1
      Contact( #O_Entrar )
      I_Contact( #Moti_ERRO )
      I_Contact( #Moti_NENC )
      I_Contact( #O_Bloqueo )
      { S7_GenerateENO := "TRUE" } Move(in := 2, out1 => #Orden_Ejecutada_Jdt)
      S_Coil( #MemoPresenciaJdt )
   END_RUNG
   RUNG wire#w1
      Contact( #O_Continuar )
      I_Contact( #Moti_ERRO )
      I_Contact( #Moti_NENC )
      I_Contact( #O_Bloqueo )
      { S7_GenerateENO := "TRUE" } Move(in := 3, out1 => #Orden_Ejecutada_Jdt)
      S_Coil( #MemoPresenciaJdt )
   END_RUNG
   RUNG wire#w1
      Contact( #O_Bloqueo )
      wire#w2
      Contact( #MX_FlujoPrin_S2 )
      { S7_GenerateENO := "TRUE" } Move(in := 12, out1 => #Orden_Ejecutada_Jdt)
      S_Coil( #MemoPresenciaJdt )
   END_RUNG
   RUNG wire#w2
      I_Contact( #MX_FlujoPrin_S2 )
      { S7_GenerateENO := "TRUE" } Move(in := 13, out1 => #Orden_Ejecutada_Jdt)
      S_Coil( #MemoPresenciaJdt )
   END_RUNG
   RUNG wire#w1
      Contact( #O_Vaciar )
      wire#w3
      Contact( #MX_FlujoPrin_S2 )
      { S7_GenerateENO := "TRUE" } Move(in := 22, out1 => #Orden_Ejecutada_Jdt)
      S_Coil( #MemoPresenciaJdt )
   END_RUNG
   RUNG wire#w3
      I_Contact( #MX_FlujoPrin_S2 )
      { S7_GenerateENO := "TRUE" } Move(in := 23, out1 => #Orden_Ejecutada_Jdt)
      S_Coil( #MemoPresenciaJdt )
   END_RUNG
   RUNG wire#w1
      I_Contact( #Habilitar_orden_JDT )
      Contact( #Moti_ERRO )
      wire#w4
      Contact( #O_Entrar )
      I_Contact( #O_Bloqueo )
      { S7_GenerateENO := "TRUE" } Move(in := 32, out1 => #Orden_Ejecutada_Jdt)
      S_Coil( #MemoPresenciaJdt )
   END_RUNG
   RUNG wire#w4
      Contact( #O_Continuar )
      I_Contact( #O_Bloqueo )
      { S7_GenerateENO := "TRUE" } Move(in := 33, out1 => #Orden_Ejecutada_Jdt)
      S_Coil( #MemoPresenciaJdt )
   END_RUNG
   RUNG wire#w1
      I_Contact( #Habilitar_orden_JDT )
      Contact( #Moti_NENC )
      wire#w5
      Contact( #O_Entrar )
      I_Contact( #O_Bloqueo )
      { S7_GenerateENO := "TRUE" } Move(in := 42, out1 => #Orden_Ejecutada_Jdt)
      S_Coil( #MemoPresenciaJdt )
   END_RUNG
   RUNG wire#w5
      Contact( #O_Continuar )
      I_Contact( #O_Bloqueo )
      { S7_GenerateENO := "TRUE" } Move(in := 43, out1 => #Orden_Ejecutada_Jdt)
      S_Coil( #MemoPresenciaJdt )
   END_RUNG
   RUNG wire#w1
      Contact( #Moti_INIC )
      wire#w6
      Contact( #O_Entrar )
      I_Contact( #O_Bloqueo )
      { S7_GenerateENO := "TRUE" } Move(in := 52, out1 => #Orden_Ejecutada_Jdt)
      S_Coil( #MemoPresenciaJdt )
   END_RUNG
   RUNG wire#w6
      Contact( #O_Continuar )
      I_Contact( #O_Bloqueo )
      { S7_GenerateENO := "TRUE" } Move(in := 53, out1 => #Orden_Ejecutada_Jdt)
      S_Coil( #MemoPresenciaJdt )
   END_RUNG
   RUNG wire#w1
      Contact( #Habilitar_orden_JDT )
      wire#w7
      Contact( #O_Entrar_JDT )
      { S7_GenerateENO := "TRUE" } Move(in := 62, out1 => #Orden_Ejecutada_Jdt)
      S_Coil( #MemoPresenciaJdt )
   END_RUNG
   RUNG wire#w7
      Contact( #O_Continuar_JDT )
      { S7_GenerateENO := "TRUE" } Move(in := 63, out1 => #Orden_Ejecutada_Jdt)
      S_Coil( #MemoPresenciaJdt )
   END_RUNG
   // the same network as SCL:
   // ENO of a box is taken as its EN; it also drops when the box reports an error
   #_w1 := NOT #T1_ET20 AND #FN_ET20;   // falling edge
   #FN_ET20 := #T1_ET20;
   IF #_w1 THEN #Etiqueta_Jdt := #Datos_Scanner.Identificador; END_IF;
   IF #_w1 AND #O_Entrar AND NOT #Moti_ERRO AND NOT #Moti_NENC AND NOT #O_Bloqueo THEN
       #Orden_Ejecutada_Jdt := 2;
       #MemoPresenciaJdt := TRUE;
   END_IF;
   IF #_w1 AND #O_Continuar AND NOT #Moti_ERRO AND NOT #Moti_NENC AND NOT #O_Bloqueo THEN
       #Orden_Ejecutada_Jdt := 3;
       #MemoPresenciaJdt := TRUE;
   END_IF;
   #_w2 := #_w1 AND #O_Bloqueo;
   IF #_w2 AND #MX_FlujoPrin_S2 THEN
       #Orden_Ejecutada_Jdt := 12;
       #MemoPresenciaJdt := TRUE;
   END_IF;
   IF #_w2 AND NOT #MX_FlujoPrin_S2 THEN
       #Orden_Ejecutada_Jdt := 13;
       #MemoPresenciaJdt := TRUE;
   END_IF;
   #_w3 := #_w1 AND #O_Vaciar;
   IF #_w3 AND #MX_FlujoPrin_S2 THEN
       #Orden_Ejecutada_Jdt := 22;
       #MemoPresenciaJdt := TRUE;
   END_IF;
   IF #_w3 AND NOT #MX_FlujoPrin_S2 THEN
       #Orden_Ejecutada_Jdt := 23;
       #MemoPresenciaJdt := TRUE;
   END_IF;
   #_w4 := #_w1 AND NOT #Habilitar_orden_JDT AND #Moti_ERRO;
   IF #_w4 AND #O_Entrar AND NOT #O_Bloqueo THEN
       #Orden_Ejecutada_Jdt := 32;
       #MemoPresenciaJdt := TRUE;
   END_IF;
   IF #_w4 AND #O_Continuar AND NOT #O_Bloqueo THEN
       #Orden_Ejecutada_Jdt := 33;
       #MemoPresenciaJdt := TRUE;
   END_IF;
   #_w5 := #_w1 AND NOT #Habilitar_orden_JDT AND #Moti_NENC;
   IF #_w5 AND #O_Entrar AND NOT #O_Bloqueo THEN
       #Orden_Ejecutada_Jdt := 42;
       #MemoPresenciaJdt := TRUE;
   END_IF;
   IF #_w5 AND #O_Continuar AND NOT #O_Bloqueo THEN
       #Orden_Ejecutada_Jdt := 43;
       #MemoPresenciaJdt := TRUE;
   END_IF;
   #_w6 := #_w1 AND #Moti_INIC;
   IF #_w6 AND #O_Entrar AND NOT #O_Bloqueo THEN
       #Orden_Ejecutada_Jdt := 52;
       #MemoPresenciaJdt := TRUE;
   END_IF;
   IF #_w6 AND #O_Continuar AND NOT #O_Bloqueo THEN
       #Orden_Ejecutada_Jdt := 53;
       #MemoPresenciaJdt := TRUE;
   END_IF;
   #_w7 := #_w1 AND #Habilitar_orden_JDT;
   IF #_w7 AND #O_Entrar_JDT THEN
       #Orden_Ejecutada_Jdt := 62;
       #MemoPresenciaJdt := TRUE;
   END_IF;
   IF #_w7 AND #O_Continuar_JDT THEN
       #Orden_Ejecutada_Jdt := 63;
       #MemoPresenciaJdt := TRUE;
   END_IF;
END_REGION

REGION Network 62: PASAR ETIQUETA JDT
   RUNG wire#powerrail
      Contact( #F_EnvMens_Mx )
      R_Coil( #MemoPresenciaJdt )
   END_RUNG
   // the same network as SCL:
   IF #F_EnvMens_Mx THEN #MemoPresenciaJdt := FALSE; END_IF;
END_REGION

REGION Network 63: PRESENCIA JDT
   RUNG wire#powerrail
      Contact( #MemoPresenciaJdt )
      Coil( #P_EnvMens_PMx )
   END_RUNG
   // the same network as SCL:
   #P_EnvMens_PMx := #MemoPresenciaJdt;
END_REGION

REGION Network 64: BORRADO ORDEN JDT
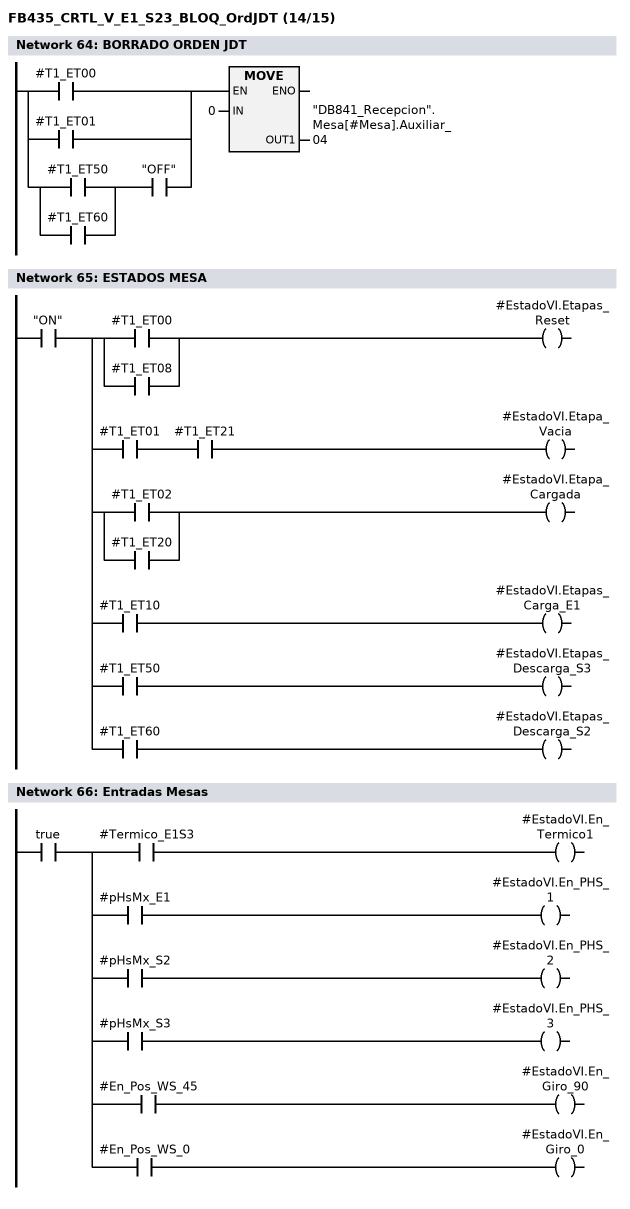
   RUNG wire#powerrail
      Contact( #T1_ET00 )
      wire#w1
      { S7_GenerateENO := "TRUE" } Move(in := 0, out1 => "DB841_Recepcion".Mesa[#Mesa].Auxiliar_04)
   END_RUNG
   RUNG wire#powerrail
      Contact( #T1_ET01 )
   END_RUNG wire#w1
   RUNG wire#powerrail
      Contact( #T1_ET50 )
      wire#w2
      Contact( "OFF" )
   END_RUNG wire#w1
   RUNG wire#powerrail
      Contact( #T1_ET60 )
   END_RUNG wire#w2
   // the same network as SCL:
   IF #T1_ET00 OR #T1_ET01 OR ((#T1_ET50 OR #T1_ET60) AND "OFF") THEN
       "DB841_Recepcion".Mesa[#Mesa].Auxiliar_04 := 0;
   END_IF;
END_REGION

REGION Network 65: ESTADOS MESA
   RUNG wire#powerrail
      Contact( "ON" )
      wire#w1
      Contact( #T1_ET00 )
      wire#w2
      Coil( #EstadoVI.Etapas_Reset )
   END_RUNG
   RUNG wire#w1
      Contact( #T1_ET08 )
   END_RUNG wire#w2
   RUNG wire#w1
      Contact( #T1_ET01 )
      Contact( #T1_ET21 )
      Coil( #EstadoVI.Etapa_Vacia )
   END_RUNG
   RUNG wire#w1
      Contact( #T1_ET02 )
      wire#w3
      Coil( #EstadoVI.Etapa_Cargada )
   END_RUNG
   RUNG wire#w1
      Contact( #T1_ET20 )
   END_RUNG wire#w3
   RUNG wire#w1
      Contact( #T1_ET10 )
      Coil( #EstadoVI.Etapas_Carga_E1 )
   END_RUNG
   RUNG wire#w1
      Contact( #T1_ET50 )
      Coil( #EstadoVI.Etapas_Descarga_S3 )
   END_RUNG
   RUNG wire#w1
      Contact( #T1_ET60 )
      Coil( #EstadoVI.Etapas_Descarga_S2 )
   END_RUNG
   // the same network as SCL:
   #EstadoVI.Etapas_Reset := "ON" AND (#T1_ET00 OR #T1_ET08);
   #EstadoVI.Etapa_Vacia := "ON" AND #T1_ET01 AND #T1_ET21;
   #EstadoVI.Etapa_Cargada := "ON" AND (#T1_ET02 OR #T1_ET20);
   #EstadoVI.Etapas_Carga_E1 := "ON" AND #T1_ET10;
   #EstadoVI.Etapas_Descarga_S3 := "ON" AND #T1_ET50;
   #EstadoVI.Etapas_Descarga_S2 := "ON" AND #T1_ET60;
END_REGION

REGION Network 66: Entradas Mesas
   RUNG wire#powerrail
      Contact( true )
      wire#w1
      Contact( #Termico_E1S3 )
      Coil( #EstadoVI.En_Termico1 )
   END_RUNG
   RUNG wire#w1
      Contact( #pHsMx_E1 )
      Coil( #EstadoVI.En_PHS_1 )
   END_RUNG
   RUNG wire#w1
      Contact( #pHsMx_S2 )
      Coil( #EstadoVI.En_PHS_2 )
   END_RUNG
   RUNG wire#w1
      Contact( #pHsMx_S3 )
      Coil( #EstadoVI.En_PHS_3 )
   END_RUNG
   RUNG wire#w1
      Contact( #En_Pos_WS_45 )
      Coil( #EstadoVI.En_Giro_90 )
   END_RUNG
   RUNG wire#w1
      Contact( #En_Pos_WS_0 )
      Coil( #EstadoVI.En_Giro_0 )
   END_RUNG
   // the same network as SCL:
   #EstadoVI.En_Termico1 := true AND #Termico_E1S3;
   #EstadoVI.En_PHS_1 := true AND #pHsMx_E1;
   #EstadoVI.En_PHS_2 := true AND #pHsMx_S2;
   #EstadoVI.En_PHS_3 := true AND #pHsMx_S3;
   #EstadoVI.En_Giro_90 := true AND #En_Pos_WS_45;
   #EstadoVI.En_Giro_0 := true AND #En_Pos_WS_0;
END_REGION

REGION Network 67: Salidas Mesas
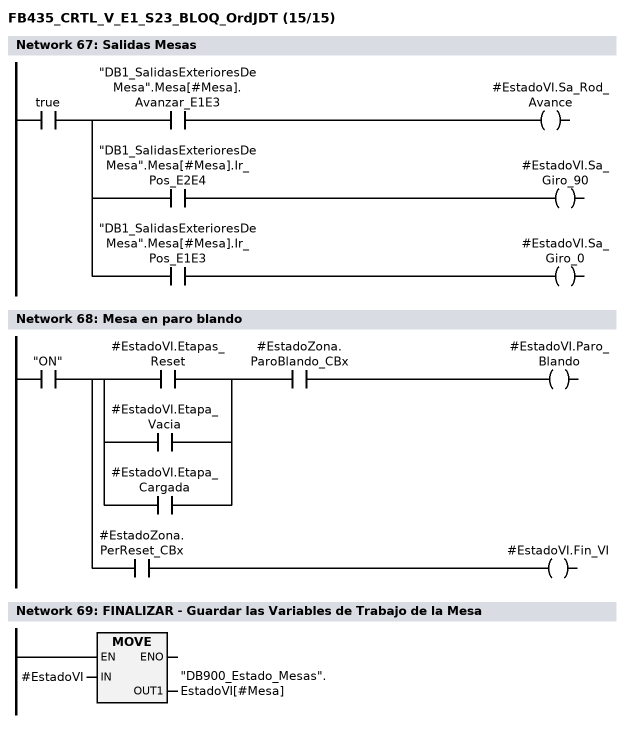
   RUNG wire#powerrail
      Contact( true )
      wire#w1
      Contact( "DB1_SalidasExterioresDeMesa".Mesa[#Mesa].Avanzar_E1E3 )
      Coil( #EstadoVI.Sa_Rod_Avance )
   END_RUNG
   RUNG wire#w1
      Contact( "DB1_SalidasExterioresDeMesa".Mesa[#Mesa].Ir_Pos_E2E4 )
      Coil( #EstadoVI.Sa_Giro_90 )
   END_RUNG
   RUNG wire#w1
      Contact( "DB1_SalidasExterioresDeMesa".Mesa[#Mesa].Ir_Pos_E1E3 )
      Coil( #EstadoVI.Sa_Giro_0 )
   END_RUNG
   // the same network as SCL:
   #EstadoVI.Sa_Rod_Avance := true AND "DB1_SalidasExterioresDeMesa".Mesa[#Mesa].Avanzar_E1E3;
   #EstadoVI.Sa_Giro_90 := true AND "DB1_SalidasExterioresDeMesa".Mesa[#Mesa].Ir_Pos_E2E4;
   #EstadoVI.Sa_Giro_0 := true AND "DB1_SalidasExterioresDeMesa".Mesa[#Mesa].Ir_Pos_E1E3;
END_REGION

REGION Network 68: Mesa en paro blando
   RUNG wire#powerrail
      Contact( "ON" )
      wire#w1
      Contact( #EstadoVI.Etapas_Reset )
      wire#w2
      Contact( #EstadoZona.ParoBlando_CBx )
      Coil( #EstadoVI.Paro_Blando )
   END_RUNG
   RUNG wire#w1
      Contact( #EstadoVI.Etapa_Vacia )
   END_RUNG wire#w2
   RUNG wire#w1
      Contact( #EstadoVI.Etapa_Cargada )
   END_RUNG wire#w2
   RUNG wire#w1
      Contact( #EstadoZona.PerReset_CBx )
      Coil( #EstadoVI.Fin_VI )
   END_RUNG
   // the same network as SCL:
   #EstadoVI.Paro_Blando := "ON" AND (#EstadoVI.Etapas_Reset OR #EstadoVI.Etapa_Vacia OR #EstadoVI.Etapa_Cargada) AND #EstadoZona.ParoBlando_CBx;
   #EstadoVI.Fin_VI := "ON" AND #EstadoZona.PerReset_CBx;
END_REGION

REGION Network 69: FINALIZAR - Guardar las Variables de Trabajo de la Mesa
   RUNG wire#powerrail
      Move(in := #EstadoVI, out1 => "DB900_Estado_Mesas".EstadoVI[#Mesa])
   END_RUNG
   // the same network as SCL:
   "DB900_Estado_Mesas".EstadoVI[#Mesa] := #EstadoVI;
END_REGION
END_FUNCTION_BLOCK
